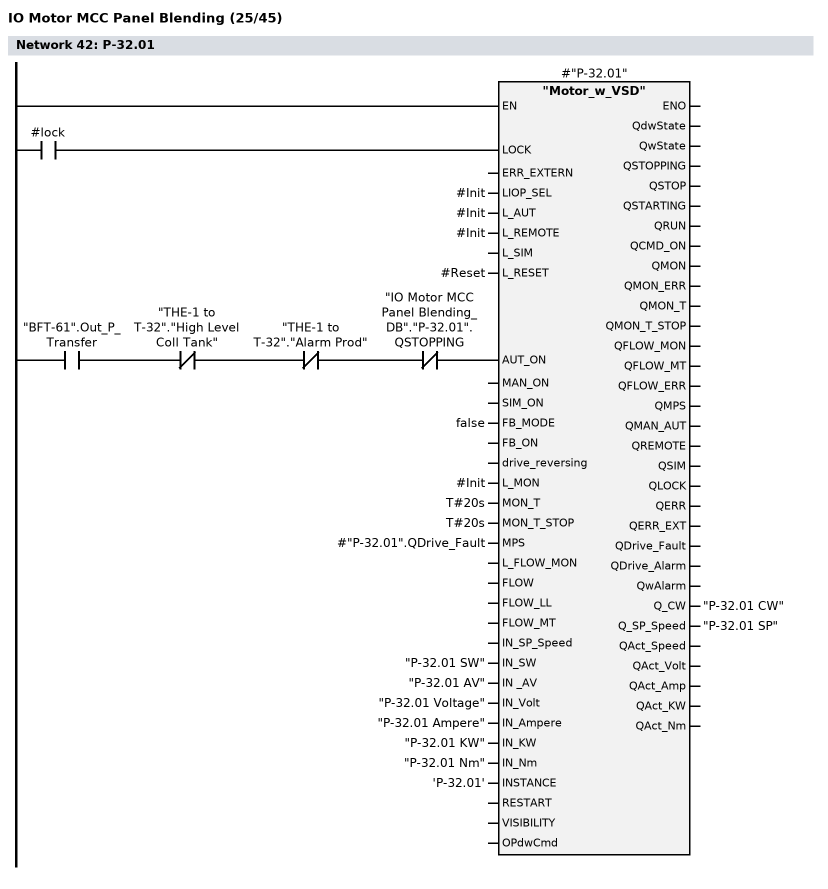
   RUNG wire#powerrail
      #"P-32.01"(LOCK := wire#w1, AUT_ON := wire#w2, ERR_EXTERN :=, LIOP_SEL := #Init, L_AUT := #Init, L_REMOTE := #Init, L_SIM :=, L_RESET := #Reset, MAN_ON :=, SIM_ON :=, FB_MODE := false, FB_ON :=, drive_reversing :=, L_MON := #Init, MON_T := T#20s, MON_T_STOP := T#20s, MPS := #"P-32.01".QDrive_Fault, L_FLOW_MON :=, FLOW :=, FLOW_LL :=, FLOW_MT :=, IN_SP_Speed :=, IN_SW := "P-32.01 SW", "IN _AV" := "P-32.01 AV", IN_Volt := "P-32.01 Voltage", IN_Ampere := "P-32.01 Ampere", IN_KW := "P-32.01 KW", IN_Nm := "P-32.01 Nm", INSTANCE := 'P-32.01', RESTART :=, VISIBILITY :=, OPdwCmd :=, QdwState =>, QwState =>, QSTOPPING =>, QSTOP =>, QSTARTING =>, QRUN =>, QCMD_ON =>, QMON =>, QMON_ERR =>, QMON_T =>, QMON_T_STOP =>, QFLOW_MON =>, QFLOW_MT =>, QFLOW_ERR =>, QMPS =>, QMAN_AUT =>, QREMOTE =>, QSIM =>, QLOCK =>, QERR =>, QERR_EXT =>, QDrive_Fault =>, QDrive_Alarm =>, QwAlarm =>, Q_CW => "P-32.01 CW", Q_SP_Speed => "P-32.01 SP", QAct_Speed =>, QAct_Volt =>, QAct_Amp =>, QAct_KW =>, QAct_Nm =>)
   END_RUNG
   RUNG wire#powerrail
      Contact( #lock )
   END_RUNG wire#w1
   RUNG wire#powerrail
      Contact( "BFT-61".Out_P_Transfer )
      I_Contact( "THE-1 to T-32"."High Level Coll Tank" )
      I_Contact( "THE-1 to T-32"."Alarm Prod" )
      I_Contact( "IO Motor MCC Panel Blending_DB"."P-32.01".QSTOPPING )
   END_RUNG wire#w2
   // the same network as SCL:
   #"P-32.01"(LOCK := #lock,   // "Motor_w_VSD"
              LIOP_SEL := #Init,
              L_AUT := #Init,
              L_REMOTE := #Init,
              L_RESET := #Reset,
              AUT_ON := "BFT-61".Out_P_Transfer AND NOT "THE-1 to T-32"."High Level Coll Tank" AND NOT "THE-1 to T-32"."Alarm Prod" AND NOT "IO Motor MCC Panel Blending_DB"."P-32.01".QSTOPPING,
              FB_MODE := false,
              L_MON := #Init,
              MON_T := T#20s,
              MON_T_STOP := T#20s,
              MPS := #"P-32.01".QDrive_Fault,
              IN_SW := "P-32.01 SW",
              "IN _AV" := "P-32.01 AV",
              IN_Volt := "P-32.01 Voltage",
              IN_Ampere := "P-32.01 Ampere",
              IN_KW := "P-32.01 KW",
              IN_Nm := "P-32.01 Nm",
              INSTANCE := 'P-32.01',
              Q_CW => "P-32.01 CW",
              Q_SP_Speed => "P-32.01 SP");
END_REGION

REGION Network 43: P-32.02
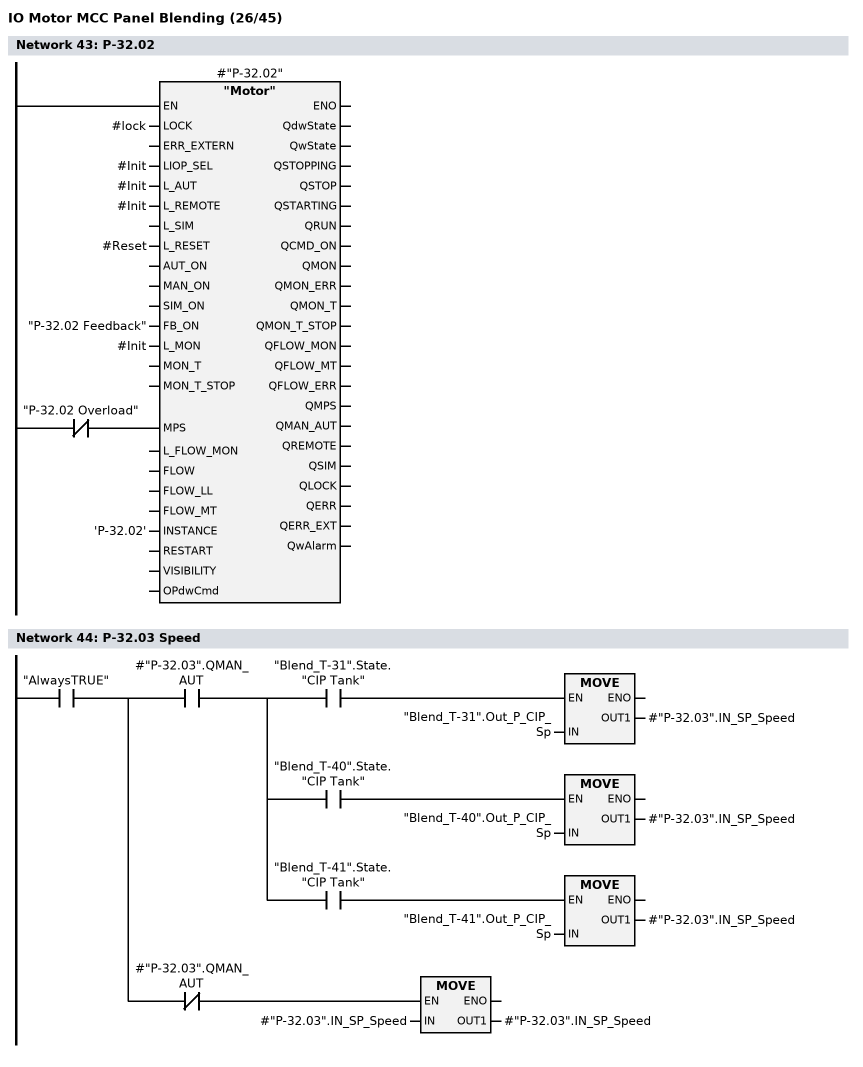
   RUNG wire#powerrail
      #"P-32.02"(MPS := wire#w1, LOCK := #lock, ERR_EXTERN :=, LIOP_SEL := #Init, L_AUT := #Init, L_REMOTE := #Init, L_SIM :=, L_RESET := #Reset, AUT_ON :=, MAN_ON :=, SIM_ON :=, FB_ON := "P-32.02 Feedback", L_MON := #Init, MON_T :=, MON_T_STOP :=, L_FLOW_MON :=, FLOW :=, FLOW_LL :=, FLOW_MT :=, INSTANCE := 'P-32.02', RESTART :=, VISIBILITY :=, OPdwCmd :=, QdwState =>, QwState =>, QSTOPPING =>, QSTOP =>, QSTARTING =>, QRUN =>, QCMD_ON =>, QMON =>, QMON_ERR =>, QMON_T =>, QMON_T_STOP =>, QFLOW_MON =>, QFLOW_MT =>, QFLOW_ERR =>, QMPS =>, QMAN_AUT =>, QREMOTE =>, QSIM =>, QLOCK =>, QERR =>, QERR_EXT =>, QwAlarm =>)
   END_RUNG
   RUNG wire#powerrail
      I_Contact( "P-32.02 Overload" )
   END_RUNG wire#w1
   // the same network as SCL:
   #"P-32.02"(LOCK := #lock,   // "Motor"
              LIOP_SEL := #Init,
              L_AUT := #Init,
              L_REMOTE := #Init,
              L_RESET := #Reset,
              FB_ON := "P-32.02 Feedback",
              L_MON := #Init,
              MPS := NOT "P-32.02 Overload",
              INSTANCE := 'P-32.02');
END_REGION

REGION Network 44: P-32.03 Speed
   RUNG wire#powerrail
      Contact( "AlwaysTRUE" )
      wire#w1
      Contact( #"P-32.03".QMAN_AUT )
      wire#w2
      Contact( "Blend_T-31".State."CIP Tank" )
      Move(in := "Blend_T-31".Out_P_CIP_Sp, out1 => #"P-32.03".IN_SP_Speed)
   END_RUNG
   RUNG wire#w2
      Contact( "Blend_T-40".State."CIP Tank" )
      Move(in := "Blend_T-40".Out_P_CIP_Sp, out1 => #"P-32.03".IN_SP_Speed)
   END_RUNG
   RUNG wire#w2
      Contact( "Blend_T-41".State."CIP Tank" )
      Move(in := "Blend_T-41".Out_P_CIP_Sp, out1 => #"P-32.03".IN_SP_Speed)
   END_RUNG
   RUNG wire#w1
      I_Contact( #"P-32.03".QMAN_AUT )
      Move(in := #"P-32.03".IN_SP_Speed, out1 => #"P-32.03".IN_SP_Speed)
   END_RUNG
   // the same network as SCL:
   #_w1 := "AlwaysTRUE" AND #"P-32.03".QMAN_AUT;
   IF #_w1 AND "Blend_T-31".State."CIP Tank" THEN
       #"P-32.03".IN_SP_Speed := "Blend_T-31".Out_P_CIP_Sp;
   END_IF;
   IF #_w1 AND "Blend_T-40".State."CIP Tank" THEN
       #"P-32.03".IN_SP_Speed := "Blend_T-40".Out_P_CIP_Sp;
   END_IF;
   IF #_w1 AND "Blend_T-41".State."CIP Tank" THEN
       #"P-32.03".IN_SP_Speed := "Blend_T-41".Out_P_CIP_Sp;
   END_IF;
   IF "AlwaysTRUE" AND NOT #"P-32.03".QMAN_AUT THEN #"P-32.03".IN_SP_Speed := #"P-32.03".IN_SP_Speed; END_IF;
END_REGION

REGION Network 45: P-32.03
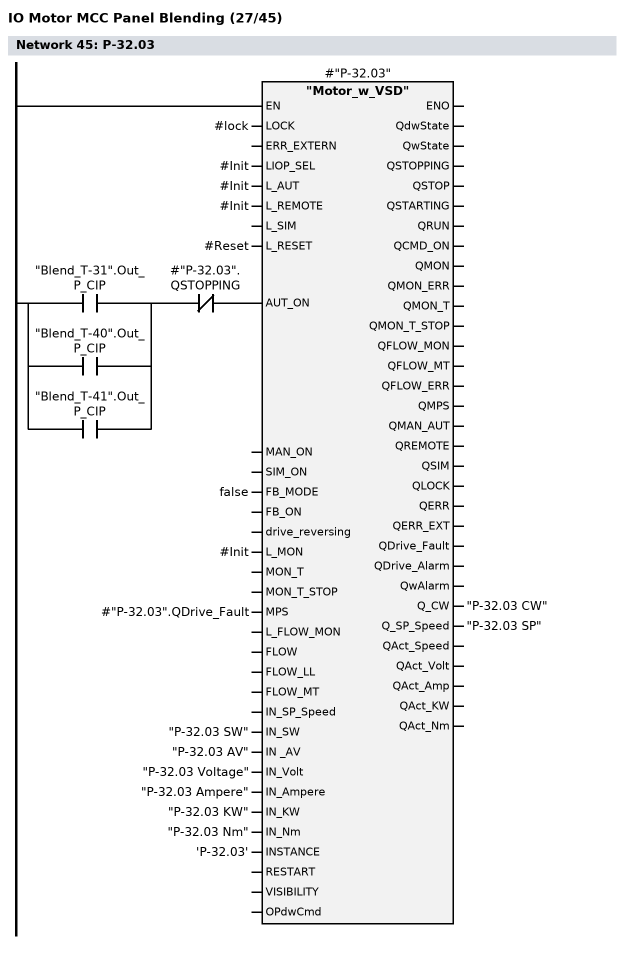
   RUNG wire#powerrail
      #"P-32.03"(AUT_ON := wire#w2, LOCK := #lock, ERR_EXTERN :=, LIOP_SEL := #Init, L_AUT := #Init, L_REMOTE := #Init, L_SIM :=, L_RESET := #Reset, MAN_ON :=, SIM_ON :=, FB_MODE := false, FB_ON :=, drive_reversing :=, L_MON := #Init, MON_T :=, MON_T_STOP :=, MPS := #"P-32.03".QDrive_Fault, L_FLOW_MON :=, FLOW :=, FLOW_LL :=, FLOW_MT :=, IN_SP_Speed :=, IN_SW := "P-32.03 SW", "IN _AV" := "P-32.03 AV", IN_Volt := "P-32.03 Voltage", IN_Ampere := "P-32.03 Ampere", IN_KW := "P-32.03 KW", IN_Nm := "P-32.03 Nm", INSTANCE := 'P-32.03', RESTART :=, VISIBILITY :=, OPdwCmd :=, QdwState =>, QwState =>, QSTOPPING =>, QSTOP =>, QSTARTING =>, QRUN =>, QCMD_ON =>, QMON =>, QMON_ERR =>, QMON_T =>, QMON_T_STOP =>, QFLOW_MON =>, QFLOW_MT =>, QFLOW_ERR =>, QMPS =>, QMAN_AUT =>, QREMOTE =>, QSIM =>, QLOCK =>, QERR =>, QERR_EXT =>, QDrive_Fault =>, QDrive_Alarm =>, QwAlarm =>, Q_CW => "P-32.03 CW", Q_SP_Speed => "P-32.03 SP", QAct_Speed =>, QAct_Volt =>, QAct_Amp =>, QAct_KW =>, QAct_Nm =>)
   END_RUNG
   RUNG wire#powerrail
      Contact( "Blend_T-31".Out_P_CIP )
      wire#w1
      I_Contact( #"P-32.03".QSTOPPING )
   END_RUNG wire#w2
   RUNG wire#powerrail
      Contact( "Blend_T-40".Out_P_CIP )
   END_RUNG wire#w1
   RUNG wire#powerrail
      Contact( "Blend_T-41".Out_P_CIP )
   END_RUNG wire#w1
   // the same network as SCL:
   #"P-32.03"(LOCK := #lock,   // "Motor_w_VSD"
              LIOP_SEL := #Init,
              L_AUT := #Init,
              L_REMOTE := #Init,
              L_RESET := #Reset,
              AUT_ON := ("Blend_T-31".Out_P_CIP OR "Blend_T-40".Out_P_CIP OR "Blend_T-41".Out_P_CIP) AND NOT #"P-32.03".QSTOPPING,
              FB_MODE := false,
              L_MON := #Init,
              MPS := #"P-32.03".QDrive_Fault,
              IN_SW := "P-32.03 SW",
              "IN _AV" := "P-32.03 AV",
              IN_Volt := "P-32.03 Voltage",
              IN_Ampere := "P-32.03 Ampere",
              IN_KW := "P-32.03 KW",
              IN_Nm := "P-32.03 Nm",
              INSTANCE := 'P-32.03',
              Q_CW => "P-32.03 CW",
              Q_SP_Speed => "P-32.03 SP");
END_REGION

REGION Network 46: P-32 Circulation (P-32.04)
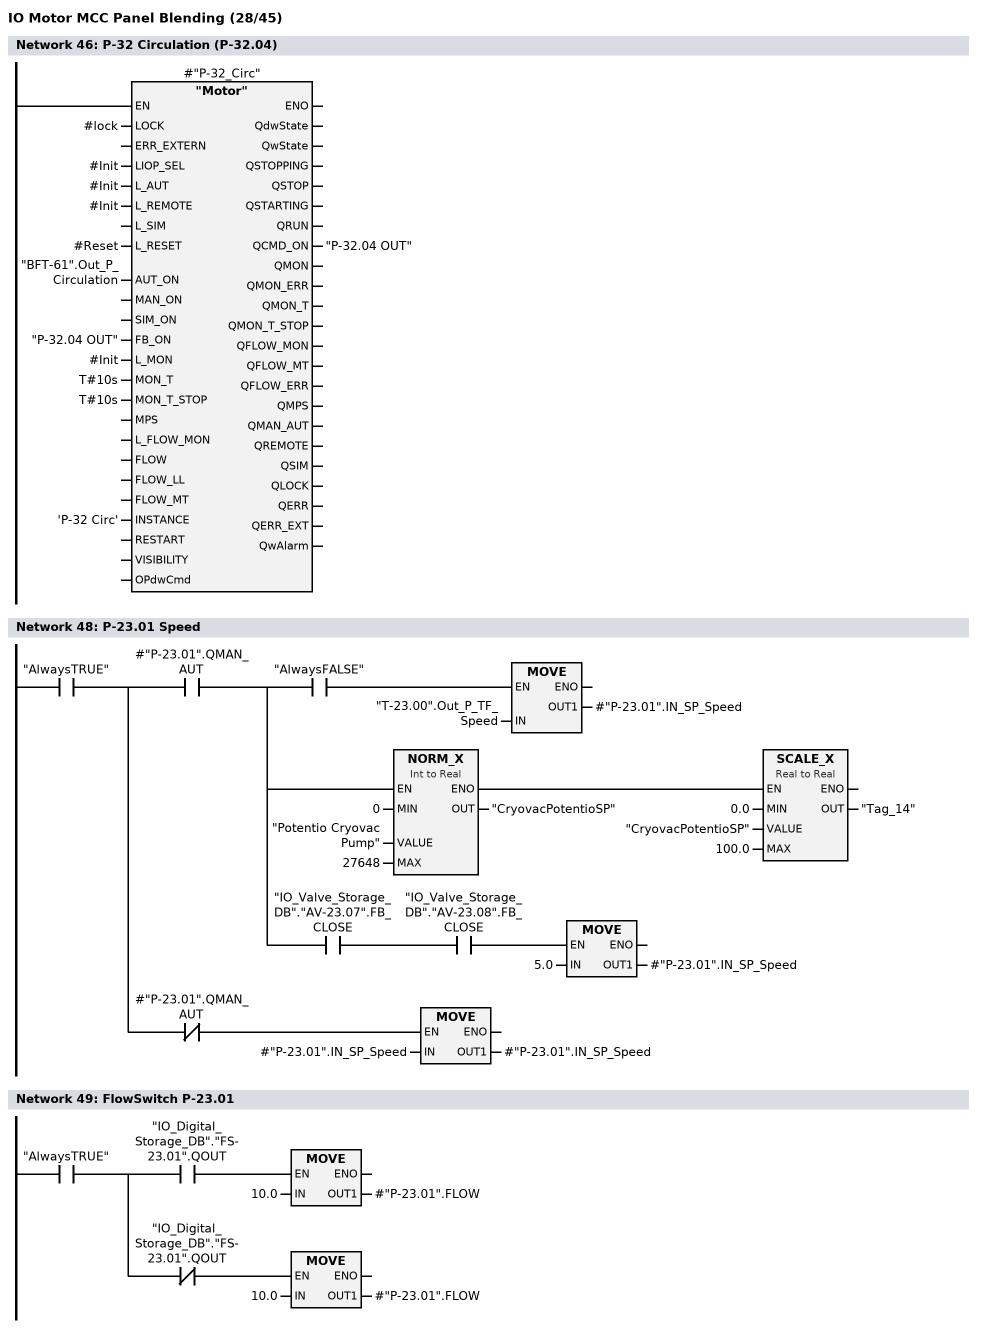
   RUNG wire#powerrail
      #"P-32_Circ"(LOCK := #lock, ERR_EXTERN :=, LIOP_SEL := #Init, L_AUT := #Init, L_REMOTE := #Init, L_SIM :=, L_RESET := #Reset, AUT_ON := "BFT-61".Out_P_Circulation, MAN_ON :=, SIM_ON :=, FB_ON := "P-32.04 OUT", L_MON := #Init, MON_T := T#10s, MON_T_STOP := T#10s, MPS :=, L_FLOW_MON :=, FLOW :=, FLOW_LL :=, FLOW_MT :=, INSTANCE := 'P-32 Circ', RESTART :=, VISIBILITY :=, OPdwCmd :=, QdwState =>, QwState =>, QSTOPPING =>, QSTOP =>, QSTARTING =>, QRUN =>, QCMD_ON => "P-32.04 OUT", QMON =>, QMON_ERR =>, QMON_T =>, QMON_T_STOP =>, QFLOW_MON =>, QFLOW_MT =>, QFLOW_ERR =>, QMPS =>, QMAN_AUT =>, QREMOTE =>, QSIM =>, QLOCK =>, QERR =>, QERR_EXT =>, QwAlarm =>)
   END_RUNG
   // the same network as SCL:
   #"P-32_Circ"(LOCK := #lock,   // "Motor"
                LIOP_SEL := #Init,
                L_AUT := #Init,
                L_REMOTE := #Init,
                L_RESET := #Reset,
                AUT_ON := "BFT-61".Out_P_Circulation,
                FB_ON := "P-32.04 OUT",
                L_MON := #Init,
                MON_T := T#10s,
                MON_T_STOP := T#10s,
                INSTANCE := 'P-32 Circ',
                QCMD_ON => "P-32.04 OUT");
END_REGION

REGION Network 48: P-23.01 Speed
   RUNG wire#powerrail
      Contact( "AlwaysTRUE" )
      wire#w1
      Contact( #"P-23.01".QMAN_AUT )
      wire#w2
      Contact( "AlwaysFALSE" )
      Move(in := "T-23.00".Out_P_TF_Speed, out1 => #"P-23.01".IN_SP_Speed)
   END_RUNG
   RUNG wire#w2
      { S7_Templates := "[SrcType := Int, DestType := Real]" } Normalize(min := 0, value := "Potentio Cryovac Pump", max := 27648, out => "CryovacPotentioSP")
      { S7_Templates := "[SrcType := Real, DestType := Real]" } Scale(min := 0.0, value := "CryovacPotentioSP", max := 100.0, out => "Tag_14")
   END_RUNG
   RUNG wire#w2
      Contact( "IO_Valve_Storage_DB"."AV-23.07".FB_CLOSE )
      Contact( "IO_Valve_Storage_DB"."AV-23.08".FB_CLOSE )
      Move(in := 5.0, out1 => #"P-23.01".IN_SP_Speed)
   END_RUNG
   RUNG wire#w1
      I_Contact( #"P-23.01".QMAN_AUT )
      Move(in := #"P-23.01".IN_SP_Speed, out1 => #"P-23.01".IN_SP_Speed)
   END_RUNG
   // the same network as SCL:
   #_w1 := "AlwaysTRUE" AND #"P-23.01".QMAN_AUT;
   IF #_w1 AND "AlwaysFALSE" THEN #"P-23.01".IN_SP_Speed := "T-23.00".Out_P_TF_Speed; END_IF;
   IF #_w1 THEN
       "CryovacPotentioSP" := NORM_X(MIN := 0, VALUE := "Potentio Cryovac Pump", MAX := 27648);
       "Tag_14" := SCALE_X(MIN := 0.0, VALUE := "CryovacPotentioSP", MAX := 100.0);
   END_IF;
   IF #_w1 AND "IO_Valve_Storage_DB"."AV-23.07".FB_CLOSE AND "IO_Valve_Storage_DB"."AV-23.08".FB_CLOSE THEN
       #"P-23.01".IN_SP_Speed := 5.0;
   END_IF;
   IF "AlwaysTRUE" AND NOT #"P-23.01".QMAN_AUT THEN #"P-23.01".IN_SP_Speed := #"P-23.01".IN_SP_Speed; END_IF;
END_REGION

REGION Network 49: FlowSwitch P-23.01
   RUNG wire#powerrail
      Contact( "AlwaysTRUE" )
      wire#w1
      Contact( "IO_Digital_Storage_DB"."FS-23.01".QOUT )
      Move(in := 10.0, out1 => #"P-23.01".FLOW)
   END_RUNG
   RUNG wire#w1
      I_Contact( "IO_Digital_Storage_DB"."FS-23.01".QOUT )
      Move(in := 10.0, out1 => #"P-23.01".FLOW)
   END_RUNG
   // the same network as SCL:
   IF "AlwaysTRUE" AND "IO_Digital_Storage_DB"."FS-23.01".QOUT THEN #"P-23.01".FLOW := 10.0; END_IF;
   IF "AlwaysTRUE" AND NOT "IO_Digital_Storage_DB"."FS-23.01".QOUT THEN #"P-23.01".FLOW := 10.0; END_IF;
END_REGION

REGION Network 50: P-23.01
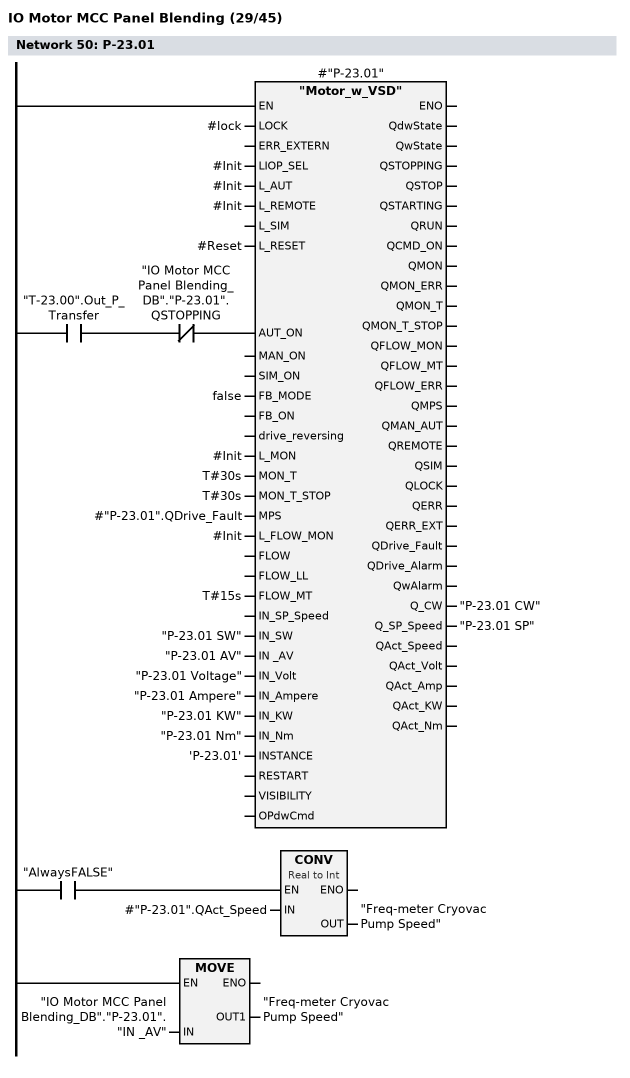
   RUNG wire#powerrail
      #"P-23.01"(AUT_ON := wire#w1, LOCK := #lock, ERR_EXTERN :=, LIOP_SEL := #Init, L_AUT := #Init, L_REMOTE := #Init, L_SIM :=, L_RESET := #Reset, MAN_ON :=, SIM_ON :=, FB_MODE := false, FB_ON :=, drive_reversing :=, L_MON := #Init, MON_T := T#30s, MON_T_STOP := T#30s, MPS := #"P-23.01".QDrive_Fault, L_FLOW_MON := #Init, FLOW :=, FLOW_LL :=, FLOW_MT := T#15s, IN_SP_Speed :=, IN_SW := "P-23.01 SW", "IN _AV" := "P-23.01 AV", IN_Volt := "P-23.01 Voltage", IN_Ampere := "P-23.01 Ampere", IN_KW := "P-23.01 KW", IN_Nm := "P-23.01 Nm", INSTANCE := 'P-23.01', RESTART :=, VISIBILITY :=, OPdwCmd :=, QdwState =>, QwState =>, QSTOPPING =>, QSTOP =>, QSTARTING =>, QRUN =>, QCMD_ON =>, QMON =>, QMON_ERR =>, QMON_T =>, QMON_T_STOP =>, QFLOW_MON =>, QFLOW_MT =>, QFLOW_ERR =>, QMPS =>, QMAN_AUT =>, QREMOTE =>, QSIM =>, QLOCK =>, QERR =>, QERR_EXT =>, QDrive_Fault =>, QDrive_Alarm =>, QwAlarm =>, Q_CW => "P-23.01 CW", Q_SP_Speed => "P-23.01 SP", QAct_Speed =>, QAct_Volt =>, QAct_Amp =>, QAct_KW =>, QAct_Nm =>)
   END_RUNG
   RUNG wire#powerrail
      Contact( "T-23.00".Out_P_Transfer )
      I_Contact( "IO Motor MCC Panel Blending_DB"."P-23.01".QSTOPPING )
   END_RUNG wire#w1
   RUNG wire#powerrail
      Contact( "AlwaysFALSE" )
      { S7_Templates := "[SrcType := Real, DestType := Int]" } Convert(in := #"P-23.01".QAct_Speed, out => "Freq-meter Cryovac Pump Speed")
   END_RUNG
   RUNG wire#powerrail
      Move(in := "IO Motor MCC Panel Blending_DB"."P-23.01"."IN _AV", out1 => "Freq-meter Cryovac Pump Speed")
   END_RUNG
   // the same network as SCL:
   #"P-23.01"(LOCK := #lock,   // "Motor_w_VSD"
              LIOP_SEL := #Init,
              L_AUT := #Init,
              L_REMOTE := #Init,
              L_RESET := #Reset,
              AUT_ON := "T-23.00".Out_P_Transfer AND NOT "IO Motor MCC Panel Blending_DB"."P-23.01".QSTOPPING,
              FB_MODE := false,
              L_MON := #Init,
              MON_T := T#30s,
              MON_T_STOP := T#30s,
              MPS := #"P-23.01".QDrive_Fault,
              L_FLOW_MON := #Init,
              FLOW_MT := T#15s,
              IN_SW := "P-23.01 SW",
              "IN _AV" := "P-23.01 AV",
              IN_Volt := "P-23.01 Voltage",
              IN_Ampere := "P-23.01 Ampere",
              IN_KW := "P-23.01 KW",
              IN_Nm := "P-23.01 Nm",
              INSTANCE := 'P-23.01',
              Q_CW => "P-23.01 CW",
              Q_SP_Speed => "P-23.01 SP");
   IF "AlwaysFALSE" THEN "Freq-meter Cryovac Pump Speed" := REAL_TO_INT(#"P-23.01".QAct_Speed); END_IF;
   "Freq-meter Cryovac Pump Speed" := "IO Motor MCC Panel Blending_DB"."P-23.01"."IN _AV";
END_REGION

REGION Network 52: P-24.01 Speed
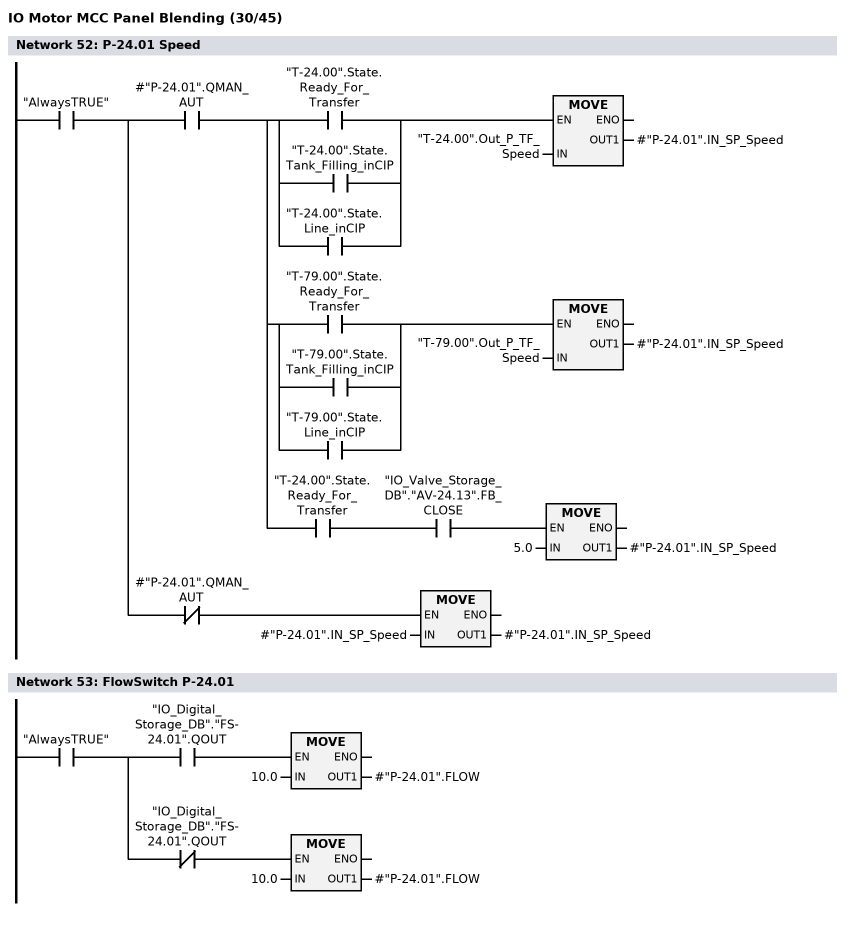
   RUNG wire#powerrail
      Contact( "AlwaysTRUE" )
      wire#w1
      Contact( #"P-24.01".QMAN_AUT )
      wire#w2
      Contact( "T-24.00".State.Ready_For_Transfer )
      wire#w3
      Move(in := "T-24.00".Out_P_TF_Speed, out1 => #"P-24.01".IN_SP_Speed)
   END_RUNG
   RUNG wire#w2
      Contact( "T-24.00".State.Tank_Filling_inCIP )
   END_RUNG wire#w3
   RUNG wire#w2
      Contact( "T-24.00".State.Line_inCIP )
   END_RUNG wire#w3
   RUNG wire#w2
      Contact( "T-79.00".State.Ready_For_Transfer )
      wire#w4
      Move(in := "T-79.00".Out_P_TF_Speed, out1 => #"P-24.01".IN_SP_Speed)
   END_RUNG
   RUNG wire#w2
      Contact( "T-79.00".State.Tank_Filling_inCIP )
   END_RUNG wire#w4
   RUNG wire#w2
      Contact( "T-79.00".State.Line_inCIP )
   END_RUNG wire#w4
   RUNG wire#w2
      Contact( "T-24.00".State.Ready_For_Transfer )
      Contact( "IO_Valve_Storage_DB"."AV-24.13".FB_CLOSE )
      Move(in := 5.0, out1 => #"P-24.01".IN_SP_Speed)
   END_RUNG
   RUNG wire#w1
      I_Contact( #"P-24.01".QMAN_AUT )
      Move(in := #"P-24.01".IN_SP_Speed, out1 => #"P-24.01".IN_SP_Speed)
   END_RUNG
   // the same network as SCL:
   #_w1 := "AlwaysTRUE" AND #"P-24.01".QMAN_AUT;
   IF #_w1 AND ("T-24.00".State.Ready_For_Transfer OR "T-24.00".State.Tank_Filling_inCIP OR "T-24.00".State.Line_inCIP) THEN
       #"P-24.01".IN_SP_Speed := "T-24.00".Out_P_TF_Speed;
   END_IF;
   IF #_w1 AND ("T-79.00".State.Ready_For_Transfer OR "T-79.00".State.Tank_Filling_inCIP OR "T-79.00".State.Line_inCIP) THEN
       #"P-24.01".IN_SP_Speed := "T-79.00".Out_P_TF_Speed;
   END_IF;
   IF #_w1 AND "T-24.00".State.Ready_For_Transfer AND "IO_Valve_Storage_DB"."AV-24.13".FB_CLOSE THEN
       #"P-24.01".IN_SP_Speed := 5.0;
   END_IF;
   IF "AlwaysTRUE" AND NOT #"P-24.01".QMAN_AUT THEN #"P-24.01".IN_SP_Speed := #"P-24.01".IN_SP_Speed; END_IF;
END_REGION

REGION Network 53: FlowSwitch P-24.01
   RUNG wire#powerrail
      Contact( "AlwaysTRUE" )
      wire#w1
      Contact( "IO_Digital_Storage_DB"."FS-24.01".QOUT )
      Move(in := 10.0, out1 => #"P-24.01".FLOW)
   END_RUNG
   RUNG wire#w1
      I_Contact( "IO_Digital_Storage_DB"."FS-24.01".QOUT )
      Move(in := 10.0, out1 => #"P-24.01".FLOW)
   END_RUNG
   // the same network as SCL:
   IF "AlwaysTRUE" AND "IO_Digital_Storage_DB"."FS-24.01".QOUT THEN #"P-24.01".FLOW := 10.0; END_IF;
   IF "AlwaysTRUE" AND NOT "IO_Digital_Storage_DB"."FS-24.01".QOUT THEN #"P-24.01".FLOW := 10.0; END_IF;
END_REGION

REGION Network 54: P-24.01
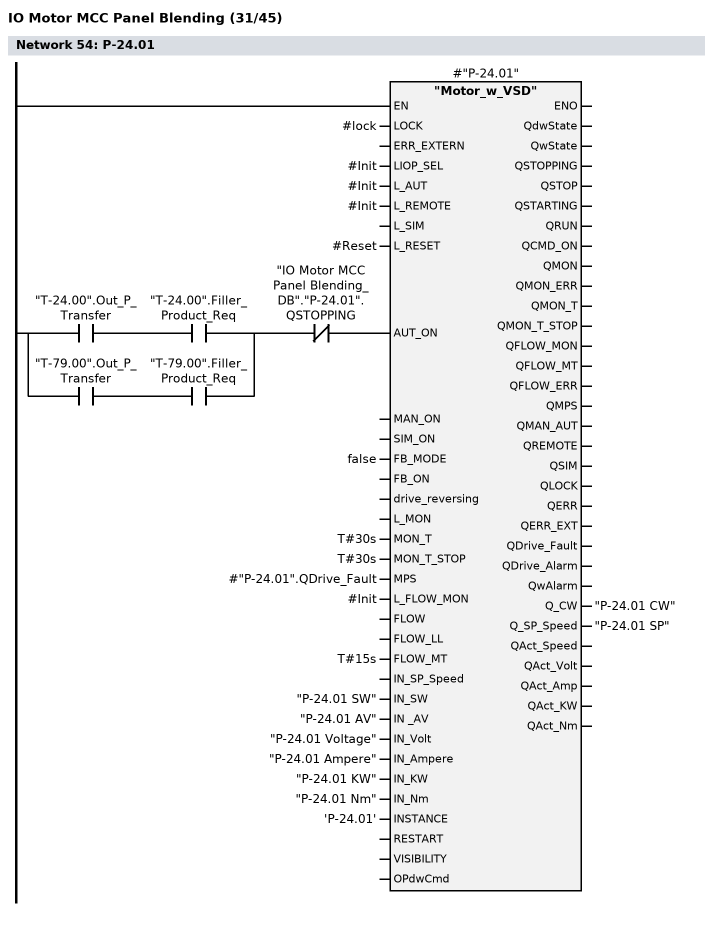
   RUNG wire#powerrail
      #"P-24.01"(AUT_ON := wire#w2, LOCK := #lock, ERR_EXTERN :=, LIOP_SEL := #Init, L_AUT := #Init, L_REMOTE := #Init, L_SIM :=, L_RESET := #Reset, MAN_ON :=, SIM_ON :=, FB_MODE := false, FB_ON :=, drive_reversing :=, L_MON :=, MON_T := T#30s, MON_T_STOP := T#30s, MPS := #"P-24.01".QDrive_Fault, L_FLOW_MON := #Init, FLOW :=, FLOW_LL :=, FLOW_MT := T#15s, IN_SP_Speed :=, IN_SW := "P-24.01 SW", "IN _AV" := "P-24.01 AV", IN_Volt := "P-24.01 Voltage", IN_Ampere := "P-24.01 Ampere", IN_KW := "P-24.01 KW", IN_Nm := "P-24.01 Nm", INSTANCE := 'P-24.01', RESTART :=, VISIBILITY :=, OPdwCmd :=, QdwState =>, QwState =>, QSTOPPING =>, QSTOP =>, QSTARTING =>, QRUN =>, QCMD_ON =>, QMON =>, QMON_ERR =>, QMON_T =>, QMON_T_STOP =>, QFLOW_MON =>, QFLOW_MT =>, QFLOW_ERR =>, QMPS =>, QMAN_AUT =>, QREMOTE =>, QSIM =>, QLOCK =>, QERR =>, QERR_EXT =>, QDrive_Fault =>, QDrive_Alarm =>, QwAlarm =>, Q_CW => "P-24.01 CW", Q_SP_Speed => "P-24.01 SP", QAct_Speed =>, QAct_Volt =>, QAct_Amp =>, QAct_KW =>, QAct_Nm =>)
   END_RUNG
   RUNG wire#powerrail
      Contact( "T-24.00".Out_P_Transfer )
      Contact( "T-24.00".Filler_Product_Req )
      wire#w1
      I_Contact( "IO Motor MCC Panel Blending_DB"."P-24.01".QSTOPPING )
   END_RUNG wire#w2
   RUNG wire#powerrail
      Contact( "T-79.00".Out_P_Transfer )
      Contact( "T-79.00".Filler_Product_Req )
   END_RUNG wire#w1
   // the same network as SCL:
   #"P-24.01"(LOCK := #lock,   // "Motor_w_VSD"
              LIOP_SEL := #Init,
              L_AUT := #Init,
              L_REMOTE := #Init,
              L_RESET := #Reset,
              AUT_ON := (("T-24.00".Out_P_Transfer AND "T-24.00".Filler_Product_Req) OR ("T-79.00".Out_P_Transfer AND "T-79.00".Filler_Product_Req)) AND NOT "IO Motor MCC Panel Blending_DB"."P-24.01".QSTOPPING,
              FB_MODE := false,
              MON_T := T#30s,
              MON_T_STOP := T#30s,
              MPS := #"P-24.01".QDrive_Fault,
              L_FLOW_MON := #Init,
              FLOW_MT := T#15s,
              IN_SW := "P-24.01 SW",
              "IN _AV" := "P-24.01 AV",
              IN_Volt := "P-24.01 Voltage",
              IN_Ampere := "P-24.01 Ampere",
              IN_KW := "P-24.01 KW",
              IN_Nm := "P-24.01 Nm",
              INSTANCE := 'P-24.01',
              Q_CW => "P-24.01 CW",
              Q_SP_Speed => "P-24.01 SP");
END_REGION

REGION Network 55: P-24.02
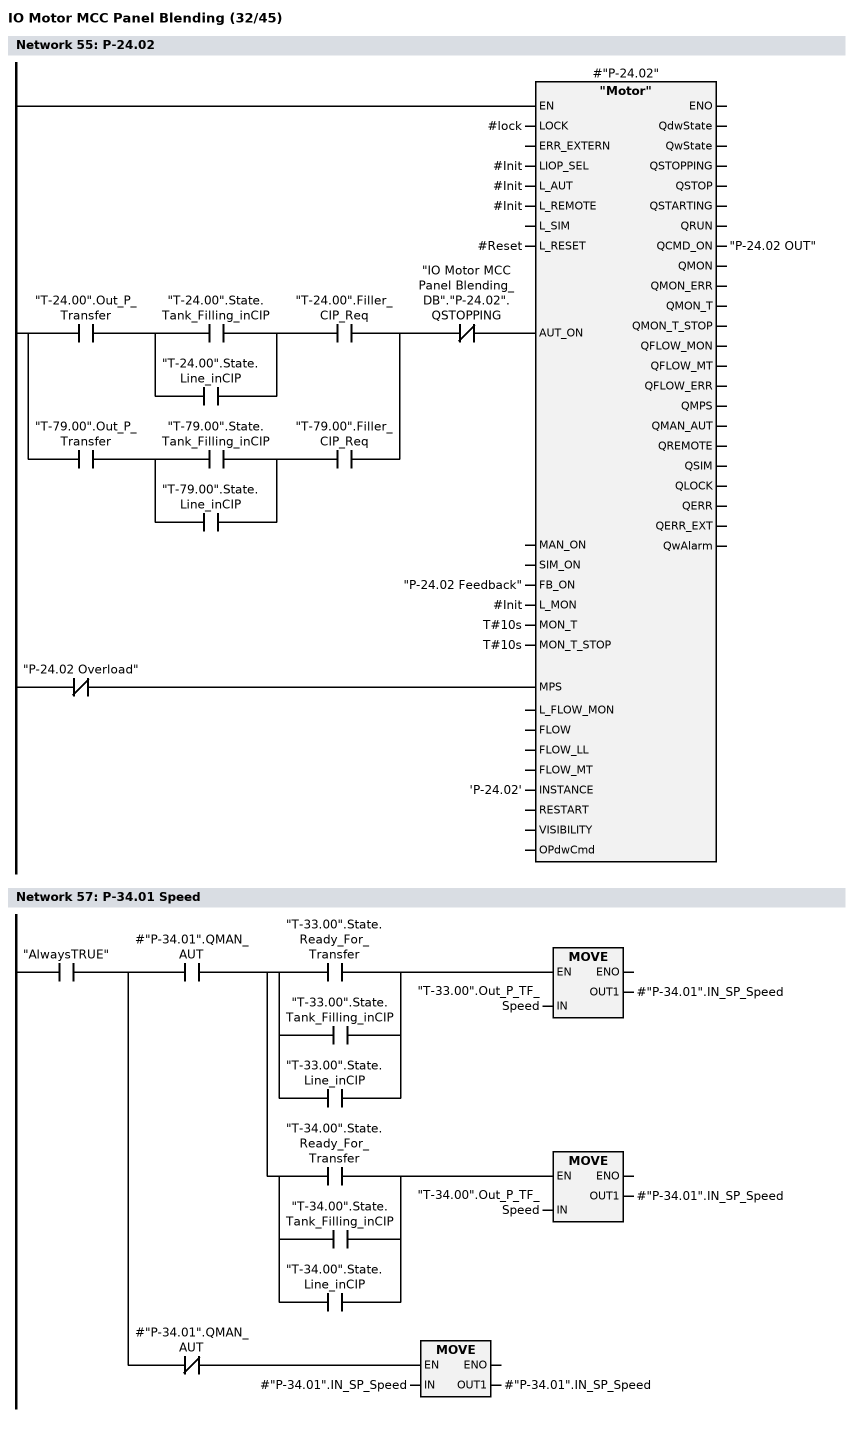
   RUNG wire#powerrail
      #"P-24.02"(AUT_ON := wire#w6, MPS := wire#w7, LOCK := #lock, ERR_EXTERN :=, LIOP_SEL := #Init, L_AUT := #Init, L_REMOTE := #Init, L_SIM :=, L_RESET := #Reset, MAN_ON :=, SIM_ON :=, FB_ON := "P-24.02 Feedback", L_MON := #Init, MON_T := T#10s, MON_T_STOP := T#10s, L_FLOW_MON :=, FLOW :=, FLOW_LL :=, FLOW_MT :=, INSTANCE := 'P-24.02', RESTART :=, VISIBILITY :=, OPdwCmd :=, QdwState =>, QwState =>, QSTOPPING =>, QSTOP =>, QSTARTING =>, QRUN =>, QCMD_ON => "P-24.02 OUT", QMON =>, QMON_ERR =>, QMON_T =>, QMON_T_STOP =>, QFLOW_MON =>, QFLOW_MT =>, QFLOW_ERR =>, QMPS =>, QMAN_AUT =>, QREMOTE =>, QSIM =>, QLOCK =>, QERR =>, QERR_EXT =>, QwAlarm =>)
   END_RUNG
   RUNG wire#powerrail
      Contact( "T-24.00".Out_P_Transfer )
      wire#w1
      Contact( "T-24.00".State.Tank_Filling_inCIP )
      wire#w2
      Contact( "T-24.00".Filler_CIP_Req )
      wire#w3
      I_Contact( "IO Motor MCC Panel Blending_DB"."P-24.02".QSTOPPING )
   END_RUNG wire#w6
   RUNG wire#w1
      Contact( "T-24.00".State.Line_inCIP )
   END_RUNG wire#w2
   RUNG wire#powerrail
      Contact( "T-79.00".Out_P_Transfer )
      wire#w4
      Contact( "T-79.00".State.Tank_Filling_inCIP )
      wire#w5
      Contact( "T-79.00".Filler_CIP_Req )
   END_RUNG wire#w3
   RUNG wire#w4
      Contact( "T-79.00".State.Line_inCIP )
   END_RUNG wire#w5
   RUNG wire#powerrail
      I_Contact( "P-24.02 Overload" )
   END_RUNG wire#w7
   // the same network as SCL:
   #"P-24.02"(LOCK := #lock,   // "Motor"
              LIOP_SEL := #Init,
              L_AUT := #Init,
              L_REMOTE := #Init,
              L_RESET := #Reset,
              AUT_ON := (("T-24.00".Out_P_Transfer AND ("T-24.00".State.Tank_Filling_inCIP OR "T-24.00".State.Line_inCIP) AND "T-24.00".Filler_CIP_Req) OR ("T-79.00".Out_P_Transfer AND ("T-79.00".State.Tank_Filling_inCIP OR "T-79.00".State.Line_inCIP) AND "T-79.00".Filler_CIP_Req)) AND NOT "IO Motor MCC Panel Blending_DB"."P-24.02".QSTOPPING,
              FB_ON := "P-24.02 Feedback",
              L_MON := #Init,
              MON_T := T#10s,
              MON_T_STOP := T#10s,
              MPS := NOT "P-24.02 Overload",
              INSTANCE := 'P-24.02',
              QCMD_ON => "P-24.02 OUT");
END_REGION

REGION Network 57: P-34.01 Speed
   RUNG wire#powerrail
      Contact( "AlwaysTRUE" )
      wire#w1
      Contact( #"P-34.01".QMAN_AUT )
      wire#w2
      Contact( "T-33.00".State.Ready_For_Transfer )
      wire#w3
      Move(in := "T-33.00".Out_P_TF_Speed, out1 => #"P-34.01".IN_SP_Speed)
   END_RUNG
   RUNG wire#w2
      Contact( "T-33.00".State.Tank_Filling_inCIP )
   END_RUNG wire#w3
   RUNG wire#w2
      Contact( "T-33.00".State.Line_inCIP )
   END_RUNG wire#w3
   RUNG wire#w2
      Contact( "T-34.00".State.Ready_For_Transfer )
      wire#w4
      Move(in := "T-34.00".Out_P_TF_Speed, out1 => #"P-34.01".IN_SP_Speed)
   END_RUNG
   RUNG wire#w2
      Contact( "T-34.00".State.Tank_Filling_inCIP )
   END_RUNG wire#w4
   RUNG wire#w2
      Contact( "T-34.00".State.Line_inCIP )
   END_RUNG wire#w4
   RUNG wire#w1
      I_Contact( #"P-34.01".QMAN_AUT )
      Move(in := #"P-34.01".IN_SP_Speed, out1 => #"P-34.01".IN_SP_Speed)
   END_RUNG
   // the same network as SCL:
   #_w1 := "AlwaysTRUE" AND #"P-34.01".QMAN_AUT;
   IF #_w1 AND ("T-33.00".State.Ready_For_Transfer OR "T-33.00".State.Tank_Filling_inCIP OR "T-33.00".State.Line_inCIP) THEN
       #"P-34.01".IN_SP_Speed := "T-33.00".Out_P_TF_Speed;
   END_IF;
   IF #_w1 AND ("T-34.00".State.Ready_For_Transfer OR "T-34.00".State.Tank_Filling_inCIP OR "T-34.00".State.Line_inCIP) THEN
       #"P-34.01".IN_SP_Speed := "T-34.00".Out_P_TF_Speed;
   END_IF;
   IF "AlwaysTRUE" AND NOT #"P-34.01".QMAN_AUT THEN #"P-34.01".IN_SP_Speed := #"P-34.01".IN_SP_Speed; END_IF;
END_REGION

REGION Network 58: FlowSwitch P-34.01
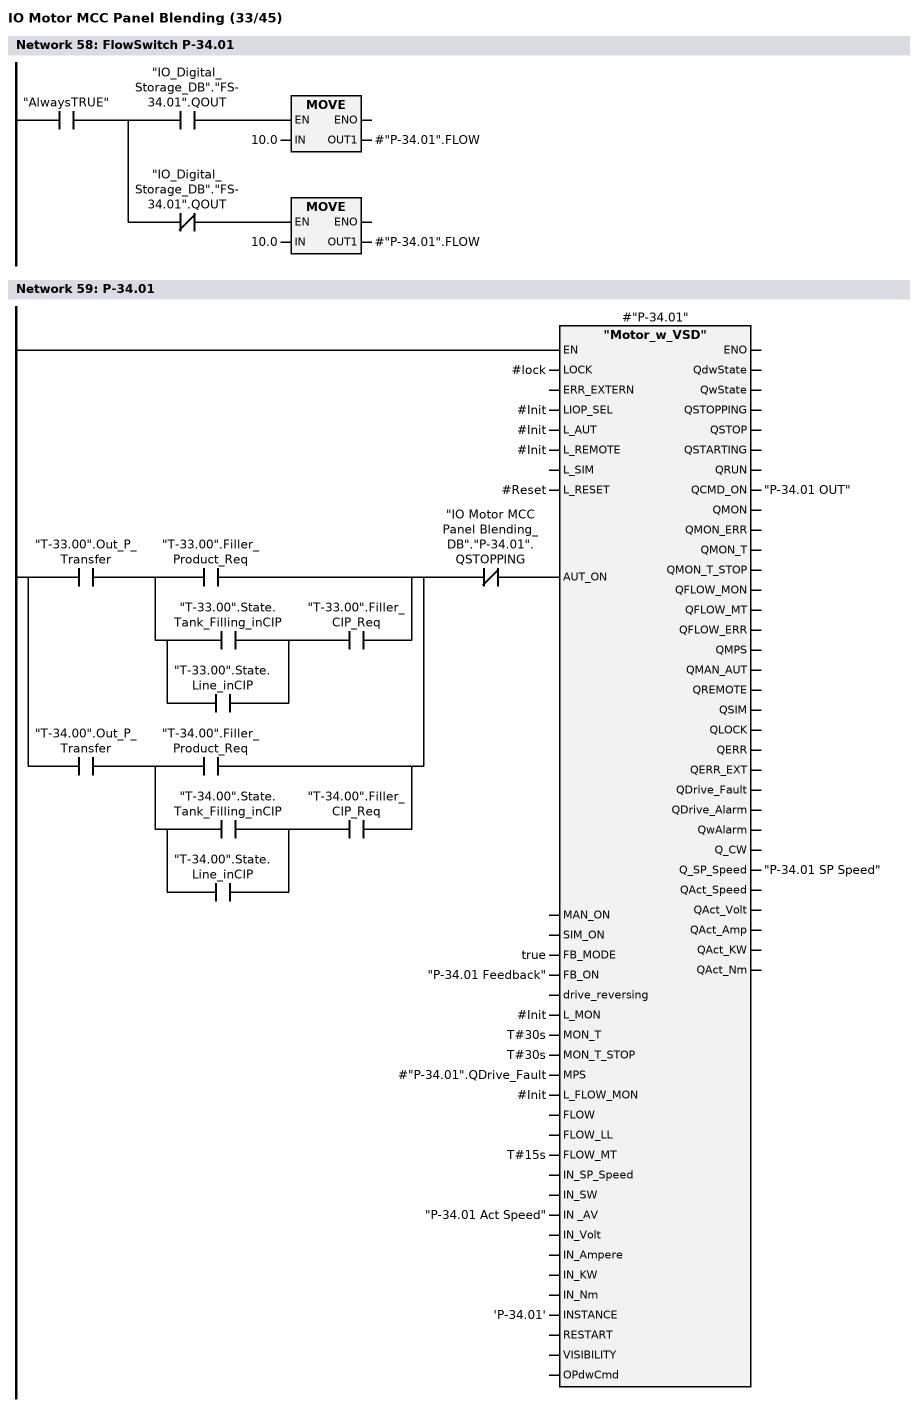
   RUNG wire#powerrail
      Contact( "AlwaysTRUE" )
      wire#w1
      Contact( "IO_Digital_Storage_DB"."FS-34.01".QOUT )
      Move(in := 10.0, out1 => #"P-34.01".FLOW)
   END_RUNG
   RUNG wire#w1
      I_Contact( "IO_Digital_Storage_DB"."FS-34.01".QOUT )
      Move(in := 10.0, out1 => #"P-34.01".FLOW)
   END_RUNG
   // the same network as SCL:
   IF "AlwaysTRUE" AND "IO_Digital_Storage_DB"."FS-34.01".QOUT THEN #"P-34.01".FLOW := 10.0; END_IF;
   IF "AlwaysTRUE" AND NOT "IO_Digital_Storage_DB"."FS-34.01".QOUT THEN #"P-34.01".FLOW := 10.0; END_IF;
END_REGION

REGION Network 59: P-34.01
   RUNG wire#powerrail
      #"P-34.01"(AUT_ON := wire#w6, LOCK := #lock, ERR_EXTERN :=, LIOP_SEL := #Init, L_AUT := #Init, L_REMOTE := #Init, L_SIM :=, L_RESET := #Reset, MAN_ON :=, SIM_ON :=, FB_MODE := true, FB_ON := "P-34.01 Feedback", drive_reversing :=, L_MON := #Init, MON_T := T#30s, MON_T_STOP := T#30s, MPS := #"P-34.01".QDrive_Fault, L_FLOW_MON := #Init, FLOW :=, FLOW_LL :=, FLOW_MT := T#15s, IN_SP_Speed :=, IN_SW :=, "IN _AV" := "P-34.01 Act Speed", IN_Volt :=, IN_Ampere :=, IN_KW :=, IN_Nm :=, INSTANCE := 'P-34.01', RESTART :=, VISIBILITY :=, OPdwCmd :=, QdwState =>, QwState =>, QSTOPPING =>, QSTOP =>, QSTARTING =>, QRUN =>, QCMD_ON => "P-34.01 OUT", QMON =>, QMON_ERR =>, QMON_T =>, QMON_T_STOP =>, QFLOW_MON =>, QFLOW_MT =>, QFLOW_ERR =>, QMPS =>, QMAN_AUT =>, QREMOTE =>, QSIM =>, QLOCK =>, QERR =>, QERR_EXT =>, QDrive_Fault =>, QDrive_Alarm =>, QwAlarm =>, Q_CW =>, Q_SP_Speed => "P-34.01 SP Speed", QAct_Speed =>, QAct_Volt =>, QAct_Amp =>, QAct_KW =>, QAct_Nm =>)
   END_RUNG
   RUNG wire#powerrail
      Contact( "T-33.00".Out_P_Transfer )
      wire#w1
      Contact( "T-33.00".Filler_Product_Req )
      wire#w2
      I_Contact( "IO Motor MCC Panel Blending_DB"."P-34.01".QSTOPPING )
   END_RUNG wire#w6
   RUNG wire#w1
      Contact( "T-33.00".State.Tank_Filling_inCIP )
      wire#w3
      Contact( "T-33.00".Filler_CIP_Req )
   END_RUNG wire#w2
   RUNG wire#w1
      Contact( "T-33.00".State.Line_inCIP )
   END_RUNG wire#w3
   RUNG wire#powerrail
      Contact( "T-34.00".Out_P_Transfer )
      wire#w4
      Contact( "T-34.00".Filler_Product_Req )
   END_RUNG wire#w2
   RUNG wire#w4
      Contact( "T-34.00".State.Tank_Filling_inCIP )
      wire#w5
      Contact( "T-34.00".Filler_CIP_Req )
   END_RUNG wire#w2
   RUNG wire#w4
      Contact( "T-34.00".State.Line_inCIP )
   END_RUNG wire#w5
   // the same network as SCL:
   #"P-34.01"(LOCK := #lock,   // "Motor_w_VSD"
              LIOP_SEL := #Init,
              L_AUT := #Init,
              L_REMOTE := #Init,
              L_RESET := #Reset,
              AUT_ON := (("T-33.00".Out_P_Transfer AND ("T-33.00".Filler_Product_Req OR (("T-33.00".State.Tank_Filling_inCIP OR "T-33.00".State.Line_inCIP) AND "T-33.00".Filler_CIP_Req))) OR ("T-34.00".Out_P_Transfer AND ("T-34.00".Filler_Product_Req OR (("T-34.00".State.Tank_Filling_inCIP OR "T-34.00".State.Line_inCIP) AND "T-34.00".Filler_CIP_Req)))) AND NOT "IO Motor MCC Panel Blending_DB"."P-34.01".QSTOPPING,
              FB_MODE := true,
              FB_ON := "P-34.01 Feedback",
              L_MON := #Init,
              MON_T := T#30s,
              MON_T_STOP := T#30s,
              MPS := #"P-34.01".QDrive_Fault,
              L_FLOW_MON := #Init,
              FLOW_MT := T#15s,
              "IN _AV" := "P-34.01 Act Speed",
              INSTANCE := 'P-34.01',
              QCMD_ON => "P-34.01 OUT",
              Q_SP_Speed => "P-34.01 SP Speed");
END_REGION

REGION Network 60: P-34.02
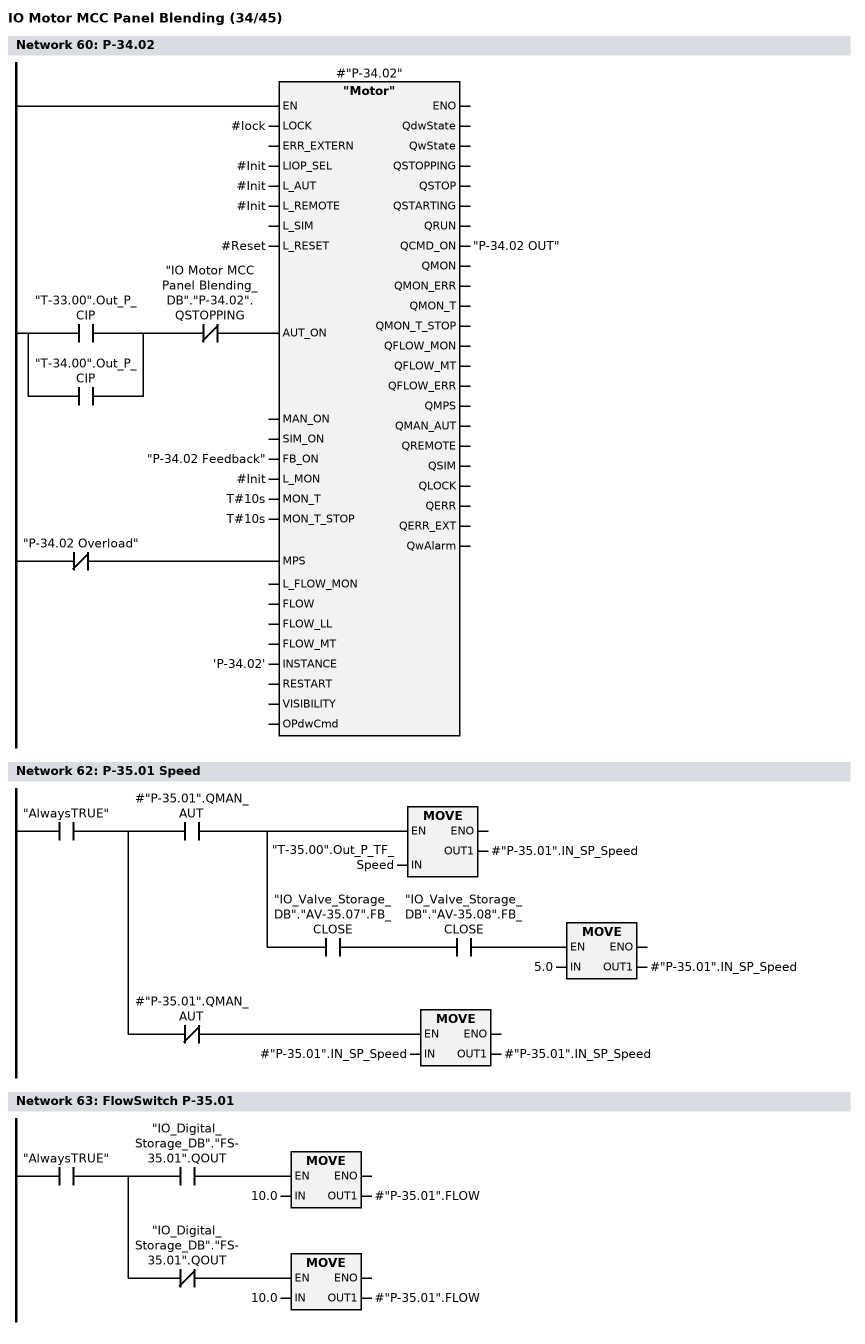
   RUNG wire#powerrail
      #"P-34.02"(AUT_ON := wire#w2, MPS := wire#w3, LOCK := #lock, ERR_EXTERN :=, LIOP_SEL := #Init, L_AUT := #Init, L_REMOTE := #Init, L_SIM :=, L_RESET := #Reset, MAN_ON :=, SIM_ON :=, FB_ON := "P-34.02 Feedback", L_MON := #Init, MON_T := T#10s, MON_T_STOP := T#10s, L_FLOW_MON :=, FLOW :=, FLOW_LL :=, FLOW_MT :=, INSTANCE := 'P-34.02', RESTART :=, VISIBILITY :=, OPdwCmd :=, QdwState =>, QwState =>, QSTOPPING =>, QSTOP =>, QSTARTING =>, QRUN =>, QCMD_ON => "P-34.02 OUT", QMON =>, QMON_ERR =>, QMON_T =>, QMON_T_STOP =>, QFLOW_MON =>, QFLOW_MT =>, QFLOW_ERR =>, QMPS =>, QMAN_AUT =>, QREMOTE =>, QSIM =>, QLOCK =>, QERR =>, QERR_EXT =>, QwAlarm =>)
   END_RUNG
   RUNG wire#powerrail
      Contact( "T-33.00".Out_P_CIP )
      wire#w1
      I_Contact( "IO Motor MCC Panel Blending_DB"."P-34.02".QSTOPPING )
   END_RUNG wire#w2
   RUNG wire#powerrail
      Contact( "T-34.00".Out_P_CIP )
   END_RUNG wire#w1
   RUNG wire#powerrail
      I_Contact( "P-34.02 Overload" )
   END_RUNG wire#w3
   // the same network as SCL:
   #"P-34.02"(LOCK := #lock,   // "Motor"
              LIOP_SEL := #Init,
              L_AUT := #Init,
              L_REMOTE := #Init,
              L_RESET := #Reset,
              AUT_ON := ("T-33.00".Out_P_CIP OR "T-34.00".Out_P_CIP) AND NOT "IO Motor MCC Panel Blending_DB"."P-34.02".QSTOPPING,
              FB_ON := "P-34.02 Feedback",
              L_MON := #Init,
              MON_T := T#10s,
              MON_T_STOP := T#10s,
              MPS := NOT "P-34.02 Overload",
              INSTANCE := 'P-34.02',
              QCMD_ON => "P-34.02 OUT");
END_REGION

REGION Network 62: P-35.01 Speed
   RUNG wire#powerrail
      Contact( "AlwaysTRUE" )
      wire#w1
      Contact( #"P-35.01".QMAN_AUT )
      wire#w2
      Move(in := "T-35.00".Out_P_TF_Speed, out1 => #"P-35.01".IN_SP_Speed)
   END_RUNG
   RUNG wire#w2
      Contact( "IO_Valve_Storage_DB"."AV-35.07".FB_CLOSE )
      Contact( "IO_Valve_Storage_DB"."AV-35.08".FB_CLOSE )
      Move(in := 5.0, out1 => #"P-35.01".IN_SP_Speed)
   END_RUNG
   RUNG wire#w1
      I_Contact( #"P-35.01".QMAN_AUT )
      Move(in := #"P-35.01".IN_SP_Speed, out1 => #"P-35.01".IN_SP_Speed)
   END_RUNG
   // the same network as SCL:
   #_w1 := "AlwaysTRUE" AND #"P-35.01".QMAN_AUT;
   IF #_w1 THEN #"P-35.01".IN_SP_Speed := "T-35.00".Out_P_TF_Speed; END_IF;
   IF #_w1 AND "IO_Valve_Storage_DB"."AV-35.07".FB_CLOSE AND "IO_Valve_Storage_DB"."AV-35.08".FB_CLOSE THEN
       #"P-35.01".IN_SP_Speed := 5.0;
   END_IF;
   IF "AlwaysTRUE" AND NOT #"P-35.01".QMAN_AUT THEN #"P-35.01".IN_SP_Speed := #"P-35.01".IN_SP_Speed; END_IF;
END_REGION

REGION Network 63: FlowSwitch P-35.01
   RUNG wire#powerrail
      Contact( "AlwaysTRUE" )
      wire#w1
      Contact( "IO_Digital_Storage_DB"."FS-35.01".QOUT )
      Move(in := 10.0, out1 => #"P-35.01".FLOW)
   END_RUNG
   RUNG wire#w1
      I_Contact( "IO_Digital_Storage_DB"."FS-35.01".QOUT )
      Move(in := 10.0, out1 => #"P-35.01".FLOW)
   END_RUNG
   // the same network as SCL:
   IF "AlwaysTRUE" AND "IO_Digital_Storage_DB"."FS-35.01".QOUT THEN #"P-35.01".FLOW := 10.0; END_IF;
   IF "AlwaysTRUE" AND NOT "IO_Digital_Storage_DB"."FS-35.01".QOUT THEN #"P-35.01".FLOW := 10.0; END_IF;
END_REGION

REGION Network 64: P-35.01
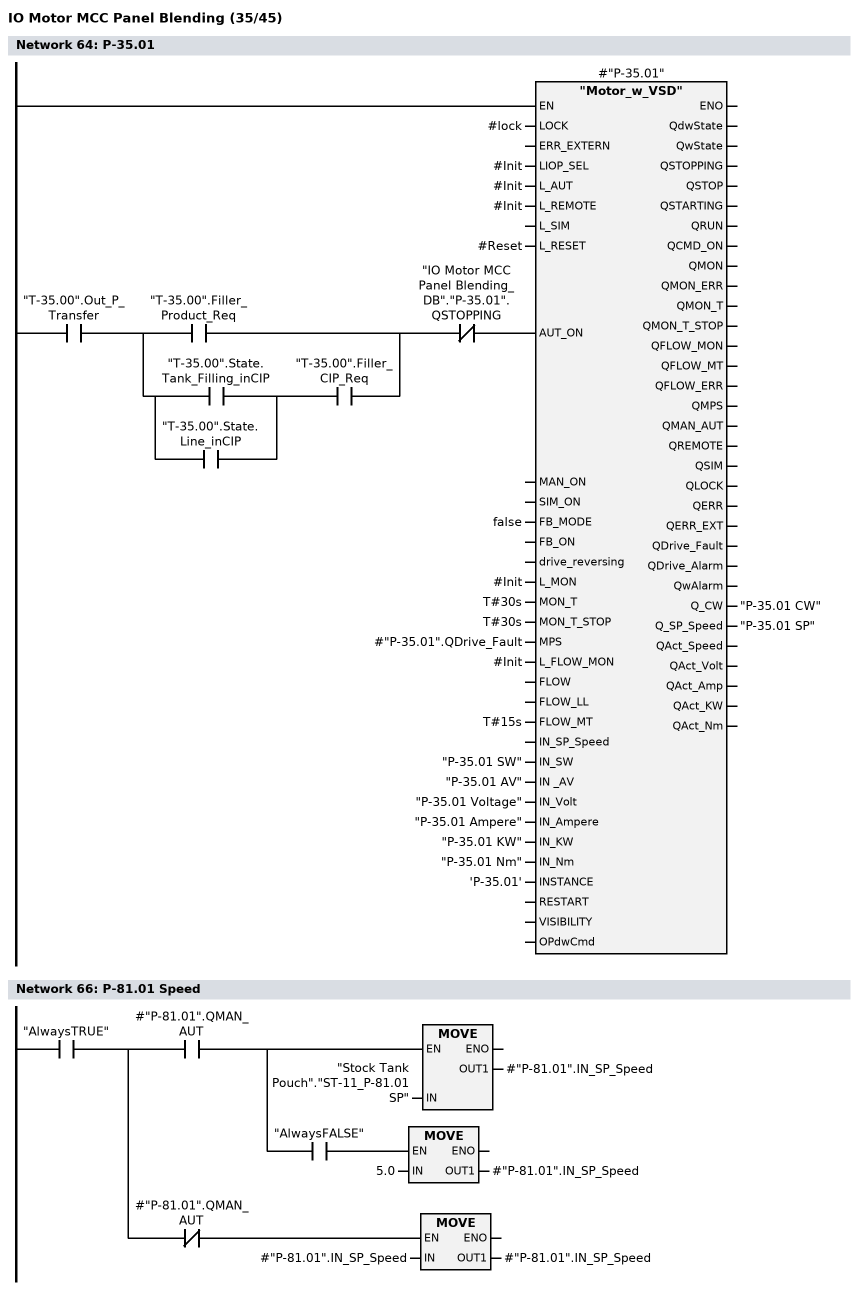
   RUNG wire#powerrail
      #"P-35.01"(AUT_ON := wire#w4, LOCK := #lock, ERR_EXTERN :=, LIOP_SEL := #Init, L_AUT := #Init, L_REMOTE := #Init, L_SIM :=, L_RESET := #Reset, MAN_ON :=, SIM_ON :=, FB_MODE := false, FB_ON :=, drive_reversing :=, L_MON := #Init, MON_T := T#30s, MON_T_STOP := T#30s, MPS := #"P-35.01".QDrive_Fault, L_FLOW_MON := #Init, FLOW :=, FLOW_LL :=, FLOW_MT := T#15s, IN_SP_Speed :=, IN_SW := "P-35.01 SW", "IN _AV" := "P-35.01 AV", IN_Volt := "P-35.01 Voltage", IN_Ampere := "P-35.01 Ampere", IN_KW := "P-35.01 KW", IN_Nm := "P-35.01 Nm", INSTANCE := 'P-35.01', RESTART :=, VISIBILITY :=, OPdwCmd :=, QdwState =>, QwState =>, QSTOPPING =>, QSTOP =>, QSTARTING =>, QRUN =>, QCMD_ON =>, QMON =>, QMON_ERR =>, QMON_T =>, QMON_T_STOP =>, QFLOW_MON =>, QFLOW_MT =>, QFLOW_ERR =>, QMPS =>, QMAN_AUT =>, QREMOTE =>, QSIM =>, QLOCK =>, QERR =>, QERR_EXT =>, QDrive_Fault =>, QDrive_Alarm =>, QwAlarm =>, Q_CW => "P-35.01 CW", Q_SP_Speed => "P-35.01 SP", QAct_Speed =>, QAct_Volt =>, QAct_Amp =>, QAct_KW =>, QAct_Nm =>)
   END_RUNG
   RUNG wire#powerrail
      Contact( "T-35.00".Out_P_Transfer )
      wire#w1
      Contact( "T-35.00".Filler_Product_Req )
      wire#w2
      I_Contact( "IO Motor MCC Panel Blending_DB"."P-35.01".QSTOPPING )
   END_RUNG wire#w4
   RUNG wire#w1
      Contact( "T-35.00".State.Tank_Filling_inCIP )
      wire#w3
      Contact( "T-35.00".Filler_CIP_Req )
   END_RUNG wire#w2
   RUNG wire#w1
      Contact( "T-35.00".State.Line_inCIP )
   END_RUNG wire#w3
   // the same network as SCL:
   #"P-35.01"(LOCK := #lock,   // "Motor_w_VSD"
              LIOP_SEL := #Init,
              L_AUT := #Init,
              L_REMOTE := #Init,
              L_RESET := #Reset,
              AUT_ON := "T-35.00".Out_P_Transfer AND ("T-35.00".Filler_Product_Req OR (("T-35.00".State.Tank_Filling_inCIP OR "T-35.00".State.Line_inCIP) AND "T-35.00".Filler_CIP_Req)) AND NOT "IO Motor MCC Panel Blending_DB"."P-35.01".QSTOPPING,
              FB_MODE := false,
              L_MON := #Init,
              MON_T := T#30s,
              MON_T_STOP := T#30s,
              MPS := #"P-35.01".QDrive_Fault,
              L_FLOW_MON := #Init,
              FLOW_MT := T#15s,
              IN_SW := "P-35.01 SW",
              "IN _AV" := "P-35.01 AV",
              IN_Volt := "P-35.01 Voltage",
              IN_Ampere := "P-35.01 Ampere",
              IN_KW := "P-35.01 KW",
              IN_Nm := "P-35.01 Nm",
              INSTANCE := 'P-35.01',
              Q_CW => "P-35.01 CW",
              Q_SP_Speed => "P-35.01 SP");
END_REGION

REGION Network 66: P-81.01 Speed
   RUNG wire#powerrail
      Contact( "AlwaysTRUE" )
      wire#w1
      Contact( #"P-81.01".QMAN_AUT )
      wire#w2
      Move(in := "Stock Tank Pouch"."ST-11_P-81.01 SP", out1 => #"P-81.01".IN_SP_Speed)
   END_RUNG
   RUNG wire#w2
      Contact( "AlwaysFALSE" )
      Move(in := 5.0, out1 => #"P-81.01".IN_SP_Speed)
   END_RUNG
   RUNG wire#w1
      I_Contact( #"P-81.01".QMAN_AUT )
      Move(in := #"P-81.01".IN_SP_Speed, out1 => #"P-81.01".IN_SP_Speed)
   END_RUNG
   // the same network as SCL:
   #_w1 := "AlwaysTRUE" AND #"P-81.01".QMAN_AUT;
   IF #_w1 THEN #"P-81.01".IN_SP_Speed := "Stock Tank Pouch"."ST-11_P-81.01 SP"; END_IF;
   IF #_w1 AND "AlwaysFALSE" THEN #"P-81.01".IN_SP_Speed := 5.0; END_IF;
   IF "AlwaysTRUE" AND NOT #"P-81.01".QMAN_AUT THEN #"P-81.01".IN_SP_Speed := #"P-81.01".IN_SP_Speed; END_IF;
END_REGION

REGION Network 67: P-81.01
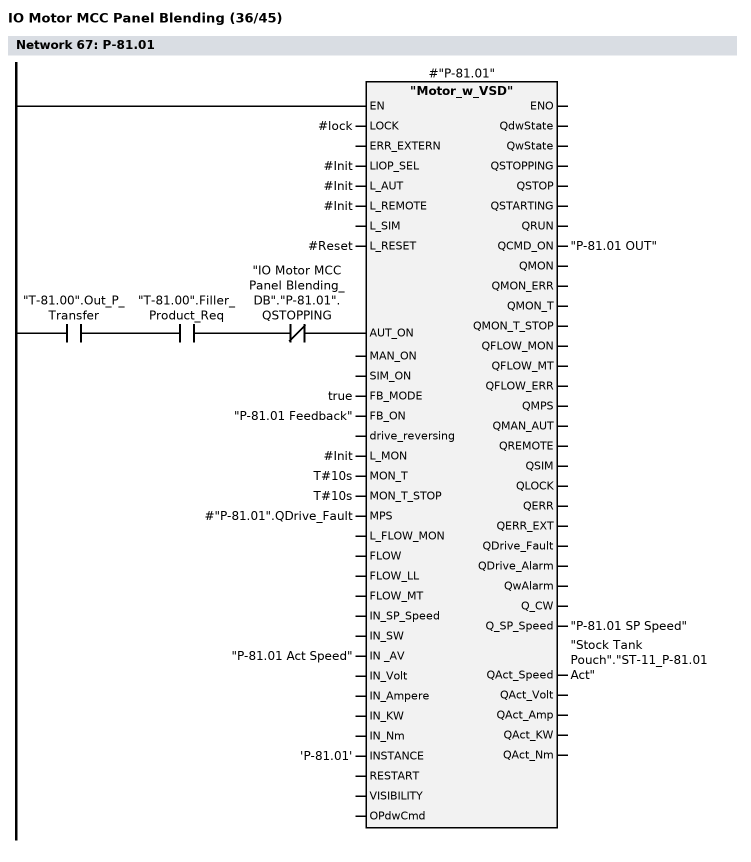
   RUNG wire#powerrail
      #"P-81.01"(AUT_ON := wire#w1, LOCK := #lock, ERR_EXTERN :=, LIOP_SEL := #Init, L_AUT := #Init, L_REMOTE := #Init, L_SIM :=, L_RESET := #Reset, MAN_ON :=, SIM_ON :=, FB_MODE := true, FB_ON := "P-81.01 Feedback", drive_reversing :=, L_MON := #Init, MON_T := T#10s, MON_T_STOP := T#10s, MPS := #"P-81.01".QDrive_Fault, L_FLOW_MON :=, FLOW :=, FLOW_LL :=, FLOW_MT :=, IN_SP_Speed :=, IN_SW :=, "IN _AV" := "P-81.01 Act Speed", IN_Volt :=, IN_Ampere :=, IN_KW :=, IN_Nm :=, INSTANCE := 'P-81.01', RESTART :=, VISIBILITY :=, OPdwCmd :=, QdwState =>, QwState =>, QSTOPPING =>, QSTOP =>, QSTARTING =>, QRUN =>, QCMD_ON => "P-81.01 OUT", QMON =>, QMON_ERR =>, QMON_T =>, QMON_T_STOP =>, QFLOW_MON =>, QFLOW_MT =>, QFLOW_ERR =>, QMPS =>, QMAN_AUT =>, QREMOTE =>, QSIM =>, QLOCK =>, QERR =>, QERR_EXT =>, QDrive_Fault =>, QDrive_Alarm =>, QwAlarm =>, Q_CW =>, Q_SP_Speed => "P-81.01 SP Speed", QAct_Speed => "Stock Tank Pouch"."ST-11_P-81.01 Act", QAct_Volt =>, QAct_Amp =>, QAct_KW =>, QAct_Nm =>)
   END_RUNG
   RUNG wire#powerrail
      Contact( "T-81.00".Out_P_Transfer )
      Contact( "T-81.00".Filler_Product_Req )
      I_Contact( "IO Motor MCC Panel Blending_DB"."P-81.01".QSTOPPING )
   END_RUNG wire#w1
   // the same network as SCL:
   #"P-81.01"(LOCK := #lock,   // "Motor_w_VSD"
              LIOP_SEL := #Init,
              L_AUT := #Init,
              L_REMOTE := #Init,
              L_RESET := #Reset,
              AUT_ON := "T-81.00".Out_P_Transfer AND "T-81.00".Filler_Product_Req AND NOT "IO Motor MCC Panel Blending_DB"."P-81.01".QSTOPPING,
              FB_MODE := true,
              FB_ON := "P-81.01 Feedback",
              L_MON := #Init,
              MON_T := T#10s,
              MON_T_STOP := T#10s,
              MPS := #"P-81.01".QDrive_Fault,
              "IN _AV" := "P-81.01 Act Speed",
              INSTANCE := 'P-81.01',
              QCMD_ON => "P-81.01 OUT",
              Q_SP_Speed => "P-81.01 SP Speed",
              QAct_Speed => "Stock Tank Pouch"."ST-11_P-81.01 Act");
END_REGION

REGION Network 68: P-81.02A
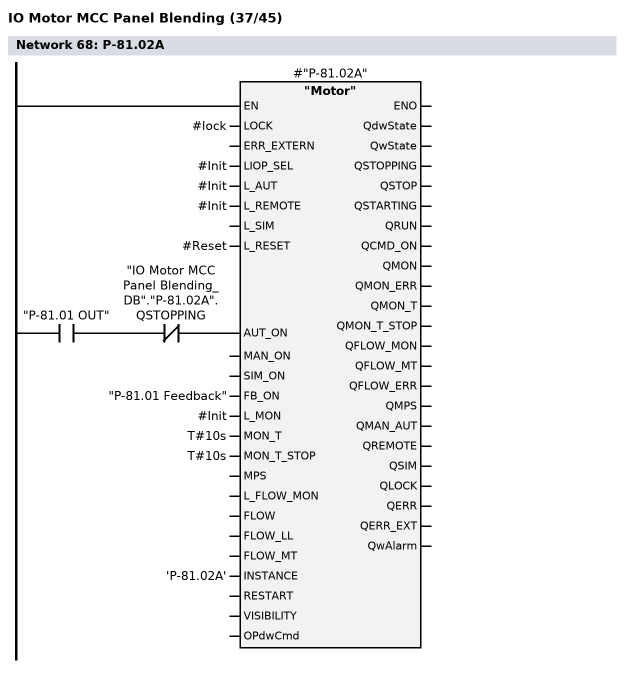
   RUNG wire#powerrail
      #"P-81.02A"(AUT_ON := wire#w1, LOCK := #lock, ERR_EXTERN :=, LIOP_SEL := #Init, L_AUT := #Init, L_REMOTE := #Init, L_SIM :=, L_RESET := #Reset, MAN_ON :=, SIM_ON :=, FB_ON := "P-81.01 Feedback", L_MON := #Init, MON_T := T#10s, MON_T_STOP := T#10s, MPS :=, L_FLOW_MON :=, FLOW :=, FLOW_LL :=, FLOW_MT :=, INSTANCE := 'P-81.02A', RESTART :=, VISIBILITY :=, OPdwCmd :=, QdwState =>, QwState =>, QSTOPPING =>, QSTOP =>, QSTARTING =>, QRUN =>, QCMD_ON =>, QMON =>, QMON_ERR =>, QMON_T =>, QMON_T_STOP =>, QFLOW_MON =>, QFLOW_MT =>, QFLOW_ERR =>, QMPS =>, QMAN_AUT =>, QREMOTE =>, QSIM =>, QLOCK =>, QERR =>, QERR_EXT =>, QwAlarm =>)
   END_RUNG
   RUNG wire#powerrail
      Contact( "P-81.01 OUT" )
      I_Contact( "IO Motor MCC Panel Blending_DB"."P-81.02A".QSTOPPING )
   END_RUNG wire#w1
   // the same network as SCL:
   #"P-81.02A"(LOCK := #lock,   // "Motor"
               LIOP_SEL := #Init,
               L_AUT := #Init,
               L_REMOTE := #Init,
               L_RESET := #Reset,
               AUT_ON := "P-81.01 OUT" AND NOT "IO Motor MCC Panel Blending_DB"."P-81.02A".QSTOPPING,
               FB_ON := "P-81.01 Feedback",
               L_MON := #Init,
               MON_T := T#10s,
               MON_T_STOP := T#10s,
               INSTANCE := 'P-81.02A');
END_REGION

REGION Network 69: P-81.02
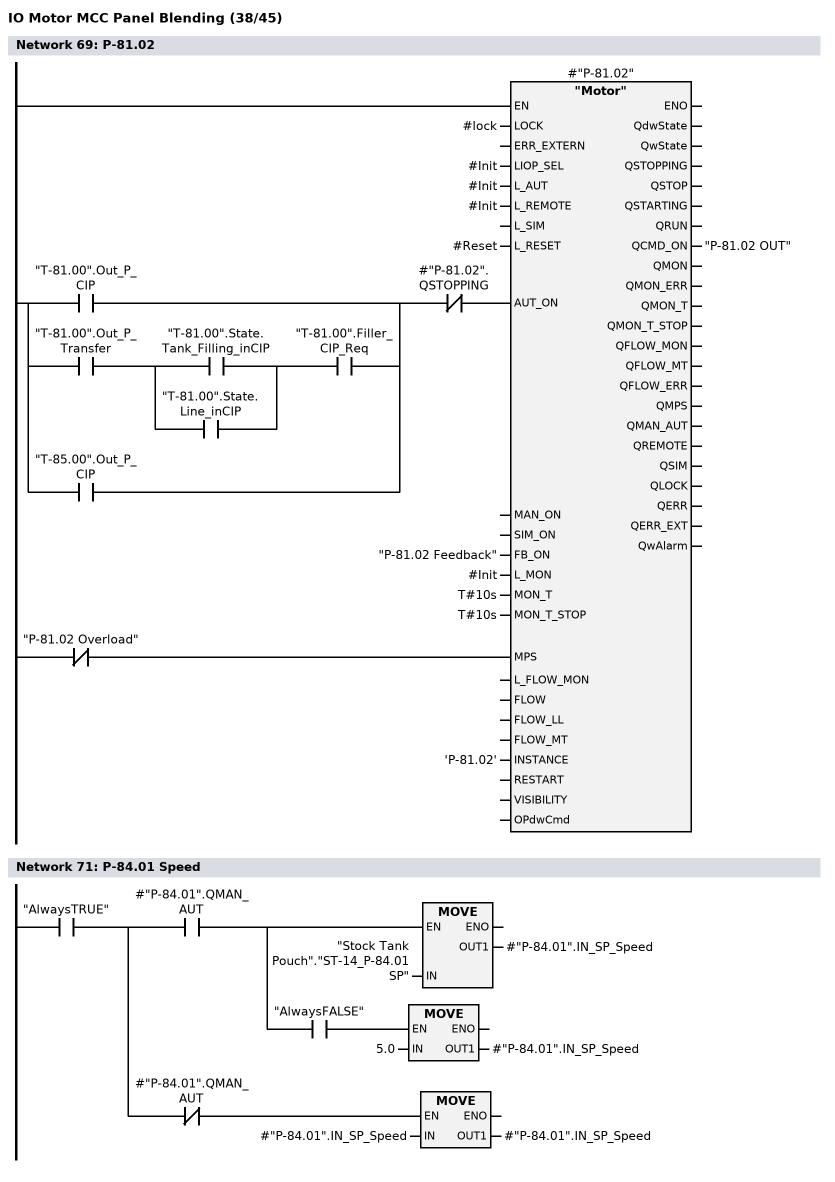
   RUNG wire#powerrail
      #"P-81.02"(AUT_ON := wire#w4, MPS := wire#w5, LOCK := #lock, ERR_EXTERN :=, LIOP_SEL := #Init, L_AUT := #Init, L_REMOTE := #Init, L_SIM :=, L_RESET := #Reset, MAN_ON :=, SIM_ON :=, FB_ON := "P-81.02 Feedback", L_MON := #Init, MON_T := T#10s, MON_T_STOP := T#10s, L_FLOW_MON :=, FLOW :=, FLOW_LL :=, FLOW_MT :=, INSTANCE := 'P-81.02', RESTART :=, VISIBILITY :=, OPdwCmd :=, QdwState =>, QwState =>, QSTOPPING =>, QSTOP =>, QSTARTING =>, QRUN =>, QCMD_ON => "P-81.02 OUT", QMON =>, QMON_ERR =>, QMON_T =>, QMON_T_STOP =>, QFLOW_MON =>, QFLOW_MT =>, QFLOW_ERR =>, QMPS =>, QMAN_AUT =>, QREMOTE =>, QSIM =>, QLOCK =>, QERR =>, QERR_EXT =>, QwAlarm =>)
   END_RUNG
   RUNG wire#powerrail
      Contact( "T-81.00".Out_P_CIP )
      wire#w1
      I_Contact( #"P-81.02".QSTOPPING )
   END_RUNG wire#w4
   RUNG wire#powerrail
      Contact( "T-81.00".Out_P_Transfer )
      wire#w2
      Contact( "T-81.00".State.Tank_Filling_inCIP )
      wire#w3
      Contact( "T-81.00".Filler_CIP_Req )
   END_RUNG wire#w1
   RUNG wire#w2
      Contact( "T-81.00".State.Line_inCIP )
   END_RUNG wire#w3
   RUNG wire#powerrail
      Contact( "T-85.00".Out_P_CIP )
   END_RUNG wire#w1
   RUNG wire#powerrail
      I_Contact( "P-81.02 Overload" )
   END_RUNG wire#w5
   // the same network as SCL:
   #"P-81.02"(LOCK := #lock,   // "Motor"
              LIOP_SEL := #Init,
              L_AUT := #Init,
              L_REMOTE := #Init,
              L_RESET := #Reset,
              AUT_ON := ("T-81.00".Out_P_CIP OR ("T-81.00".Out_P_Transfer AND ("T-81.00".State.Tank_Filling_inCIP OR "T-81.00".State.Line_inCIP) AND "T-81.00".Filler_CIP_Req) OR "T-85.00".Out_P_CIP) AND NOT #"P-81.02".QSTOPPING,
              FB_ON := "P-81.02 Feedback",
              L_MON := #Init,
              MON_T := T#10s,
              MON_T_STOP := T#10s,
              MPS := NOT "P-81.02 Overload",
              INSTANCE := 'P-81.02',
              QCMD_ON => "P-81.02 OUT");
END_REGION

REGION Network 71: P-84.01 Speed
   RUNG wire#powerrail
      Contact( "AlwaysTRUE" )
      wire#w1
      Contact( #"P-84.01".QMAN_AUT )
      wire#w2
      Move(in := "Stock Tank Pouch"."ST-14_P-84.01 SP", out1 => #"P-84.01".IN_SP_Speed)
   END_RUNG
   RUNG wire#w2
      Contact( "AlwaysFALSE" )
      Move(in := 5.0, out1 => #"P-84.01".IN_SP_Speed)
   END_RUNG
   RUNG wire#w1
      I_Contact( #"P-84.01".QMAN_AUT )
      Move(in := #"P-84.01".IN_SP_Speed, out1 => #"P-84.01".IN_SP_Speed)
   END_RUNG
   // the same network as SCL:
   #_w1 := "AlwaysTRUE" AND #"P-84.01".QMAN_AUT;
   IF #_w1 THEN #"P-84.01".IN_SP_Speed := "Stock Tank Pouch"."ST-14_P-84.01 SP"; END_IF;
   IF #_w1 AND "AlwaysFALSE" THEN #"P-84.01".IN_SP_Speed := 5.0; END_IF;
   IF "AlwaysTRUE" AND NOT #"P-84.01".QMAN_AUT THEN #"P-84.01".IN_SP_Speed := #"P-84.01".IN_SP_Speed; END_IF;
END_REGION

REGION Network 72: P-84.01
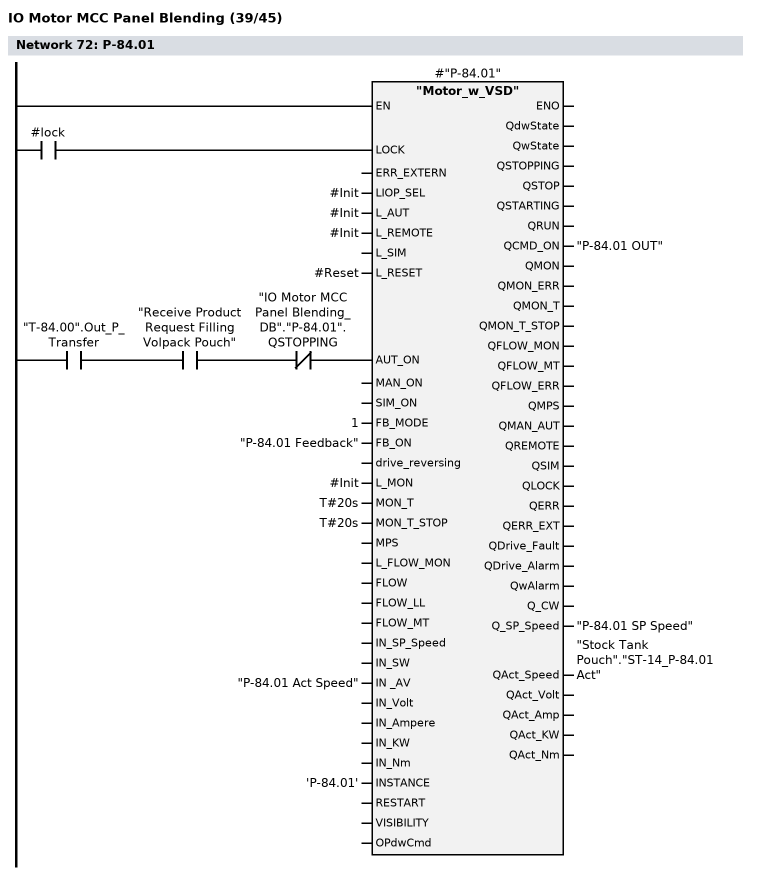
   RUNG wire#powerrail
      #"P-84.01"(LOCK := wire#w1, AUT_ON := wire#w2, ERR_EXTERN :=, LIOP_SEL := #Init, L_AUT := #Init, L_REMOTE := #Init, L_SIM :=, L_RESET := #Reset, MAN_ON :=, SIM_ON :=, FB_MODE := 1, FB_ON := "P-84.01 Feedback", drive_reversing :=, L_MON := #Init, MON_T := T#20s, MON_T_STOP := T#20s, MPS :=, L_FLOW_MON :=, FLOW :=, FLOW_LL :=, FLOW_MT :=, IN_SP_Speed :=, IN_SW :=, "IN _AV" := "P-84.01 Act Speed", IN_Volt :=, IN_Ampere :=, IN_KW :=, IN_Nm :=, INSTANCE := 'P-84.01', RESTART :=, VISIBILITY :=, OPdwCmd :=, QdwState =>, QwState =>, QSTOPPING =>, QSTOP =>, QSTARTING =>, QRUN =>, QCMD_ON => "P-84.01 OUT", QMON =>, QMON_ERR =>, QMON_T =>, QMON_T_STOP =>, QFLOW_MON =>, QFLOW_MT =>, QFLOW_ERR =>, QMPS =>, QMAN_AUT =>, QREMOTE =>, QSIM =>, QLOCK =>, QERR =>, QERR_EXT =>, QDrive_Fault =>, QDrive_Alarm =>, QwAlarm =>, Q_CW =>, Q_SP_Speed => "P-84.01 SP Speed", QAct_Speed => "Stock Tank Pouch"."ST-14_P-84.01 Act", QAct_Volt =>, QAct_Amp =>, QAct_KW =>, QAct_Nm =>)
   END_RUNG
   RUNG wire#powerrail
      Contact( #lock )
   END_RUNG wire#w1
   RUNG wire#powerrail
      Contact( "T-84.00".Out_P_Transfer )
      Contact( "Receive Product Request Filling Volpack Pouch" )
      I_Contact( "IO Motor MCC Panel Blending_DB"."P-84.01".QSTOPPING )
   END_RUNG wire#w2
   // the same network as SCL:
   #"P-84.01"(LOCK := #lock,   // "Motor_w_VSD"
              LIOP_SEL := #Init,
              L_AUT := #Init,
              L_REMOTE := #Init,
              L_RESET := #Reset,
              AUT_ON := "T-84.00".Out_P_Transfer AND "Receive Product Request Filling Volpack Pouch" AND NOT "IO Motor MCC Panel Blending_DB"."P-84.01".QSTOPPING,
              FB_MODE := 1,
              FB_ON := "P-84.01 Feedback",
              L_MON := #Init,
              MON_T := T#20s,
              MON_T_STOP := T#20s,
              "IN _AV" := "P-84.01 Act Speed",
              INSTANCE := 'P-84.01',
              QCMD_ON => "P-84.01 OUT",
              Q_SP_Speed => "P-84.01 SP Speed",
              QAct_Speed => "Stock Tank Pouch"."ST-14_P-84.01 Act");
END_REGION

REGION Network 73: P-84.01A
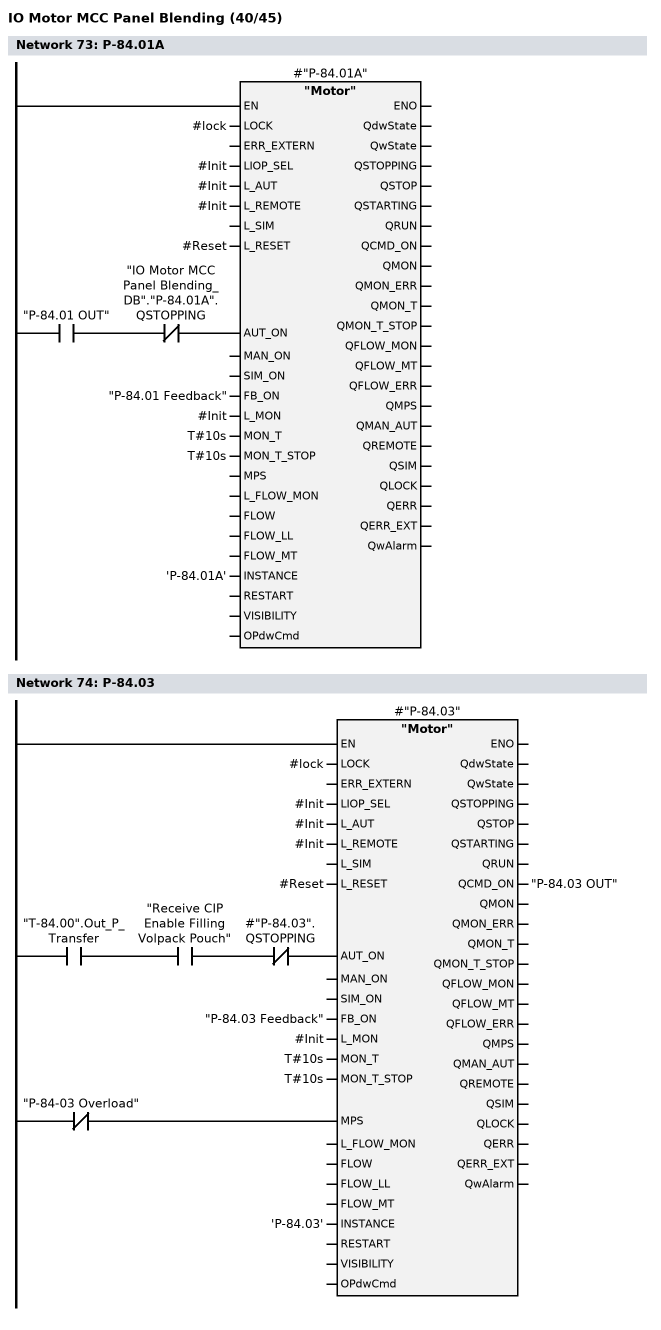
   RUNG wire#powerrail
      #"P-84.01A"(AUT_ON := wire#w1, LOCK := #lock, ERR_EXTERN :=, LIOP_SEL := #Init, L_AUT := #Init, L_REMOTE := #Init, L_SIM :=, L_RESET := #Reset, MAN_ON :=, SIM_ON :=, FB_ON := "P-84.01 Feedback", L_MON := #Init, MON_T := T#10s, MON_T_STOP := T#10s, MPS :=, L_FLOW_MON :=, FLOW :=, FLOW_LL :=, FLOW_MT :=, INSTANCE := 'P-84.01A', RESTART :=, VISIBILITY :=, OPdwCmd :=, QdwState =>, QwState =>, QSTOPPING =>, QSTOP =>, QSTARTING =>, QRUN =>, QCMD_ON =>, QMON =>, QMON_ERR =>, QMON_T =>, QMON_T_STOP =>, QFLOW_MON =>, QFLOW_MT =>, QFLOW_ERR =>, QMPS =>, QMAN_AUT =>, QREMOTE =>, QSIM =>, QLOCK =>, QERR =>, QERR_EXT =>, QwAlarm =>)
   END_RUNG
   RUNG wire#powerrail
      Contact( "P-84.01 OUT" )
      I_Contact( "IO Motor MCC Panel Blending_DB"."P-84.01A".QSTOPPING )
   END_RUNG wire#w1
   // the same network as SCL:
   #"P-84.01A"(LOCK := #lock,   // "Motor"
               LIOP_SEL := #Init,
               L_AUT := #Init,
               L_REMOTE := #Init,
               L_RESET := #Reset,
               AUT_ON := "P-84.01 OUT" AND NOT "IO Motor MCC Panel Blending_DB"."P-84.01A".QSTOPPING,
               FB_ON := "P-84.01 Feedback",
               L_MON := #Init,
               MON_T := T#10s,
               MON_T_STOP := T#10s,
               INSTANCE := 'P-84.01A');
END_REGION

REGION Network 74: P-84.03
   RUNG wire#powerrail
      #"P-84.03"(AUT_ON := wire#w1, MPS := wire#w2, LOCK := #lock, ERR_EXTERN :=, LIOP_SEL := #Init, L_AUT := #Init, L_REMOTE := #Init, L_SIM :=, L_RESET := #Reset, MAN_ON :=, SIM_ON :=, FB_ON := "P-84.03 Feedback", L_MON := #Init, MON_T := T#10s, MON_T_STOP := T#10s, L_FLOW_MON :=, FLOW :=, FLOW_LL :=, FLOW_MT :=, INSTANCE := 'P-84.03', RESTART :=, VISIBILITY :=, OPdwCmd :=, QdwState =>, QwState =>, QSTOPPING =>, QSTOP =>, QSTARTING =>, QRUN =>, QCMD_ON => "P-84.03 OUT", QMON =>, QMON_ERR =>, QMON_T =>, QMON_T_STOP =>, QFLOW_MON =>, QFLOW_MT =>, QFLOW_ERR =>, QMPS =>, QMAN_AUT =>, QREMOTE =>, QSIM =>, QLOCK =>, QERR =>, QERR_EXT =>, QwAlarm =>)
   END_RUNG
   RUNG wire#powerrail
      Contact( "T-84.00".Out_P_Transfer )
      Contact( "Receive CIP Enable Filling Volpack Pouch" )
      I_Contact( #"P-84.03".QSTOPPING )
   END_RUNG wire#w1
   RUNG wire#powerrail
      I_Contact( "P-84-03 Overload" )
   END_RUNG wire#w2
   // the same network as SCL:
   #"P-84.03"(LOCK := #lock,   // "Motor"
              LIOP_SEL := #Init,
              L_AUT := #Init,
              L_REMOTE := #Init,
              L_RESET := #Reset,
              AUT_ON := "T-84.00".Out_P_Transfer AND "Receive CIP Enable Filling Volpack Pouch" AND NOT #"P-84.03".QSTOPPING,
              FB_ON := "P-84.03 Feedback",
              L_MON := #Init,
              MON_T := T#10s,
              MON_T_STOP := T#10s,
              MPS := NOT "P-84-03 Overload",
              INSTANCE := 'P-84.03',
              QCMD_ON => "P-84.03 OUT");
END_REGION

REGION Network 75: P-84.02 Speed
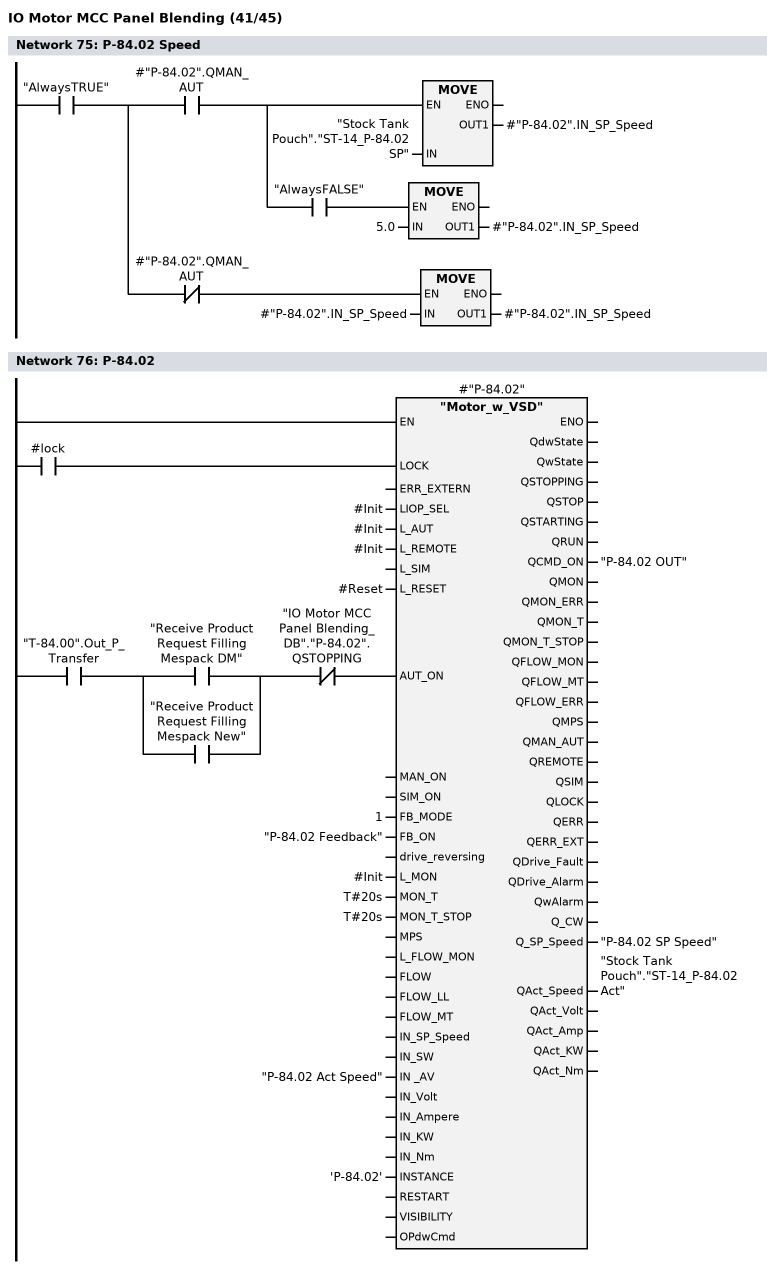
   RUNG wire#powerrail
      Contact( "AlwaysTRUE" )
      wire#w1
      Contact( #"P-84.02".QMAN_AUT )
      wire#w2
      Move(in := "Stock Tank Pouch"."ST-14_P-84.02 SP", out1 => #"P-84.02".IN_SP_Speed)
   END_RUNG
   RUNG wire#w2
      Contact( "AlwaysFALSE" )
      Move(in := 5.0, out1 => #"P-84.02".IN_SP_Speed)
   END_RUNG
   RUNG wire#w1
      I_Contact( #"P-84.02".QMAN_AUT )
      Move(in := #"P-84.02".IN_SP_Speed, out1 => #"P-84.02".IN_SP_Speed)
   END_RUNG
   // the same network as SCL:
   #_w1 := "AlwaysTRUE" AND #"P-84.02".QMAN_AUT;
   IF #_w1 THEN #"P-84.02".IN_SP_Speed := "Stock Tank Pouch"."ST-14_P-84.02 SP"; END_IF;
   IF #_w1 AND "AlwaysFALSE" THEN #"P-84.02".IN_SP_Speed := 5.0; END_IF;
   IF "AlwaysTRUE" AND NOT #"P-84.02".QMAN_AUT THEN #"P-84.02".IN_SP_Speed := #"P-84.02".IN_SP_Speed; END_IF;
END_REGION

REGION Network 76: P-84.02
   RUNG wire#powerrail
      #"P-84.02"(LOCK := wire#w1, AUT_ON := wire#w4, ERR_EXTERN :=, LIOP_SEL := #Init, L_AUT := #Init, L_REMOTE := #Init, L_SIM :=, L_RESET := #Reset, MAN_ON :=, SIM_ON :=, FB_MODE := 1, FB_ON := "P-84.02 Feedback", drive_reversing :=, L_MON := #Init, MON_T := T#20s, MON_T_STOP := T#20s, MPS :=, L_FLOW_MON :=, FLOW :=, FLOW_LL :=, FLOW_MT :=, IN_SP_Speed :=, IN_SW :=, "IN _AV" := "P-84.02 Act Speed", IN_Volt :=, IN_Ampere :=, IN_KW :=, IN_Nm :=, INSTANCE := 'P-84.02', RESTART :=, VISIBILITY :=, OPdwCmd :=, QdwState =>, QwState =>, QSTOPPING =>, QSTOP =>, QSTARTING =>, QRUN =>, QCMD_ON => "P-84.02 OUT", QMON =>, QMON_ERR =>, QMON_T =>, QMON_T_STOP =>, QFLOW_MON =>, QFLOW_MT =>, QFLOW_ERR =>, QMPS =>, QMAN_AUT =>, QREMOTE =>, QSIM =>, QLOCK =>, QERR =>, QERR_EXT =>, QDrive_Fault =>, QDrive_Alarm =>, QwAlarm =>, Q_CW =>, Q_SP_Speed => "P-84.02 SP Speed", QAct_Speed => "Stock Tank Pouch"."ST-14_P-84.02 Act", QAct_Volt =>, QAct_Amp =>, QAct_KW =>, QAct_Nm =>)
   END_RUNG
   RUNG wire#powerrail
      Contact( #lock )
   END_RUNG wire#w1
   RUNG wire#powerrail
      Contact( "T-84.00".Out_P_Transfer )
      wire#w2
      Contact( "Receive Product Request Filling Mespack DM" )
      wire#w3
      I_Contact( "IO Motor MCC Panel Blending_DB"."P-84.02".QSTOPPING )
   END_RUNG wire#w4
   RUNG wire#w2
      Contact( "Receive Product Request Filling Mespack New" )
   END_RUNG wire#w3
   // the same network as SCL:
   #"P-84.02"(LOCK := #lock,   // "Motor_w_VSD"
              LIOP_SEL := #Init,
              L_AUT := #Init,
              L_REMOTE := #Init,
              L_RESET := #Reset,
              AUT_ON := "T-84.00".Out_P_Transfer AND ("Receive Product Request Filling Mespack DM" OR "Receive Product Request Filling Mespack New") AND NOT "IO Motor MCC Panel Blending_DB"."P-84.02".QSTOPPING,
              FB_MODE := 1,
              FB_ON := "P-84.02 Feedback",
              L_MON := #Init,
              MON_T := T#20s,
              MON_T_STOP := T#20s,
              "IN _AV" := "P-84.02 Act Speed",
              INSTANCE := 'P-84.02',
              QCMD_ON => "P-84.02 OUT",
              Q_SP_Speed => "P-84.02 SP Speed",
              QAct_Speed => "Stock Tank Pouch"."ST-14_P-84.02 Act");
END_REGION

REGION Network 77: P-84.02A
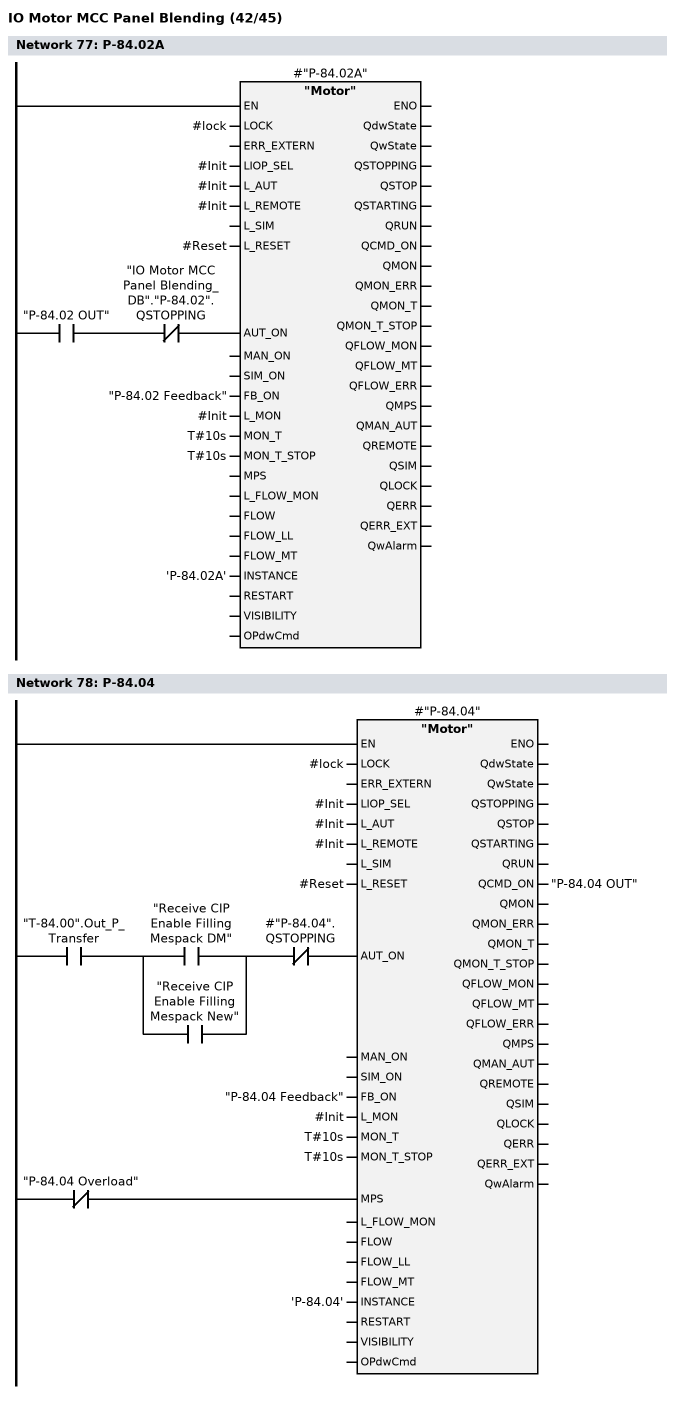
   RUNG wire#powerrail
      #"P-84.02A"(AUT_ON := wire#w1, LOCK := #lock, ERR_EXTERN :=, LIOP_SEL := #Init, L_AUT := #Init, L_REMOTE := #Init, L_SIM :=, L_RESET := #Reset, MAN_ON :=, SIM_ON :=, FB_ON := "P-84.02 Feedback", L_MON := #Init, MON_T := T#10s, MON_T_STOP := T#10s, MPS :=, L_FLOW_MON :=, FLOW :=, FLOW_LL :=, FLOW_MT :=, INSTANCE := 'P-84.02A', RESTART :=, VISIBILITY :=, OPdwCmd :=, QdwState =>, QwState =>, QSTOPPING =>, QSTOP =>, QSTARTING =>, QRUN =>, QCMD_ON =>, QMON =>, QMON_ERR =>, QMON_T =>, QMON_T_STOP =>, QFLOW_MON =>, QFLOW_MT =>, QFLOW_ERR =>, QMPS =>, QMAN_AUT =>, QREMOTE =>, QSIM =>, QLOCK =>, QERR =>, QERR_EXT =>, QwAlarm =>)
   END_RUNG
   RUNG wire#powerrail
      Contact( "P-84.02 OUT" )
      I_Contact( "IO Motor MCC Panel Blending_DB"."P-84.02".QSTOPPING )
   END_RUNG wire#w1
   // the same network as SCL:
   #"P-84.02A"(LOCK := #lock,   // "Motor"
               LIOP_SEL := #Init,
               L_AUT := #Init,
               L_REMOTE := #Init,
               L_RESET := #Reset,
               AUT_ON := "P-84.02 OUT" AND NOT "IO Motor MCC Panel Blending_DB"."P-84.02".QSTOPPING,
               FB_ON := "P-84.02 Feedback",
               L_MON := #Init,
               MON_T := T#10s,
               MON_T_STOP := T#10s,
               INSTANCE := 'P-84.02A');
END_REGION

REGION Network 78: P-84.04
   RUNG wire#powerrail
      #"P-84.04"(AUT_ON := wire#w3, MPS := wire#w4, LOCK := #lock, ERR_EXTERN :=, LIOP_SEL := #Init, L_AUT := #Init, L_REMOTE := #Init, L_SIM :=, L_RESET := #Reset, MAN_ON :=, SIM_ON :=, FB_ON := "P-84.04 Feedback", L_MON := #Init, MON_T := T#10s, MON_T_STOP := T#10s, L_FLOW_MON :=, FLOW :=, FLOW_LL :=, FLOW_MT :=, INSTANCE := 'P-84.04', RESTART :=, VISIBILITY :=, OPdwCmd :=, QdwState =>, QwState =>, QSTOPPING =>, QSTOP =>, QSTARTING =>, QRUN =>, QCMD_ON => "P-84.04 OUT", QMON =>, QMON_ERR =>, QMON_T =>, QMON_T_STOP =>, QFLOW_MON =>, QFLOW_MT =>, QFLOW_ERR =>, QMPS =>, QMAN_AUT =>, QREMOTE =>, QSIM =>, QLOCK =>, QERR =>, QERR_EXT =>, QwAlarm =>)
   END_RUNG
   RUNG wire#powerrail
      Contact( "T-84.00".Out_P_Transfer )
      wire#w1
      Contact( "Receive CIP Enable Filling Mespack DM" )
      wire#w2
      I_Contact( #"P-84.04".QSTOPPING )
   END_RUNG wire#w3
   RUNG wire#w1
      Contact( "Receive CIP Enable Filling Mespack New" )
   END_RUNG wire#w2
   RUNG wire#powerrail
      I_Contact( "P-84.04 Overload" )
   END_RUNG wire#w4
   // the same network as SCL:
   #"P-84.04"(LOCK := #lock,   // "Motor"
              LIOP_SEL := #Init,
              L_AUT := #Init,
              L_REMOTE := #Init,
              L_RESET := #Reset,
              AUT_ON := "T-84.00".Out_P_Transfer AND ("Receive CIP Enable Filling Mespack DM" OR "Receive CIP Enable Filling Mespack New") AND NOT #"P-84.04".QSTOPPING,
              FB_ON := "P-84.04 Feedback",
              L_MON := #Init,
              MON_T := T#10s,
              MON_T_STOP := T#10s,
              MPS := NOT "P-84.04 Overload",
              INSTANCE := 'P-84.04',
              QCMD_ON => "P-84.04 OUT");
END_REGION

REGION Network 80: P-82.01 Speed
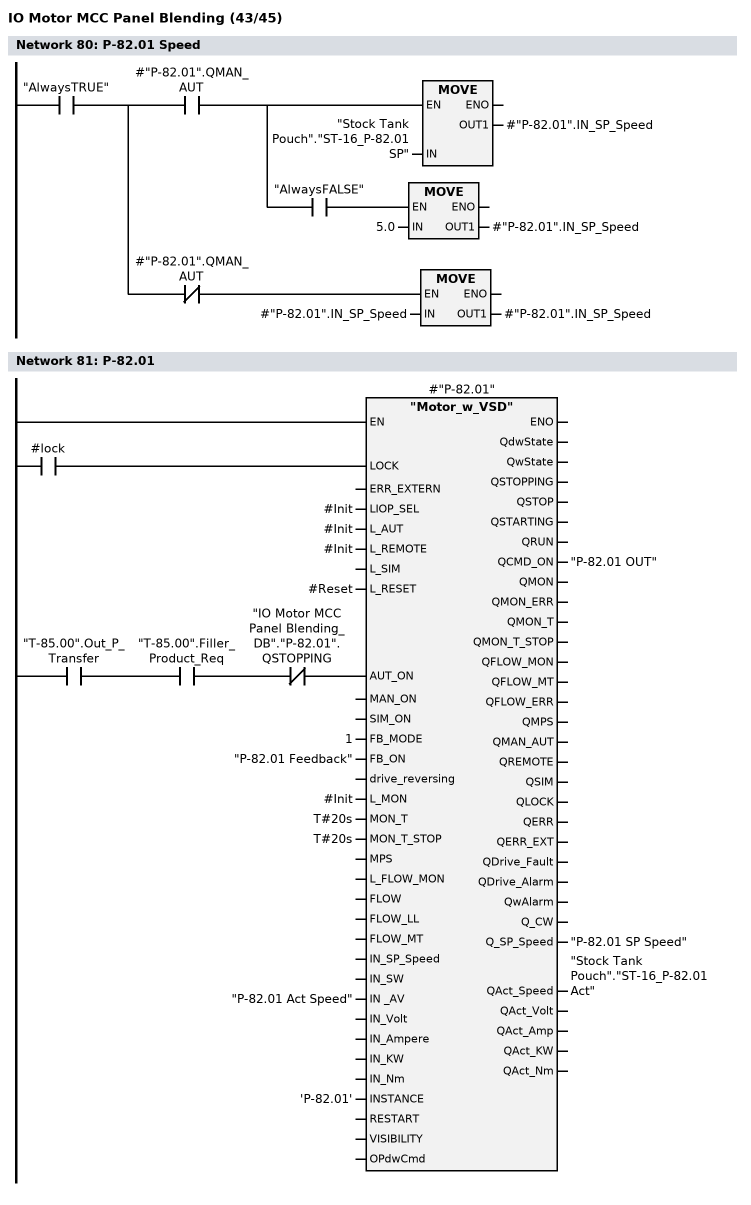
   RUNG wire#powerrail
      Contact( "AlwaysTRUE" )
      wire#w1
      Contact( #"P-82.01".QMAN_AUT )
      wire#w2
      Move(in := "Stock Tank Pouch"."ST-16_P-82.01 SP", out1 => #"P-82.01".IN_SP_Speed)
   END_RUNG
   RUNG wire#w2
      Contact( "AlwaysFALSE" )
      Move(in := 5.0, out1 => #"P-82.01".IN_SP_Speed)
   END_RUNG
   RUNG wire#w1
      I_Contact( #"P-82.01".QMAN_AUT )
      Move(in := #"P-82.01".IN_SP_Speed, out1 => #"P-82.01".IN_SP_Speed)
   END_RUNG
   // the same network as SCL:
   #_w1 := "AlwaysTRUE" AND #"P-82.01".QMAN_AUT;
   IF #_w1 THEN #"P-82.01".IN_SP_Speed := "Stock Tank Pouch"."ST-16_P-82.01 SP"; END_IF;
   IF #_w1 AND "AlwaysFALSE" THEN #"P-82.01".IN_SP_Speed := 5.0; END_IF;
   IF "AlwaysTRUE" AND NOT #"P-82.01".QMAN_AUT THEN #"P-82.01".IN_SP_Speed := #"P-82.01".IN_SP_Speed; END_IF;
END_REGION

REGION Network 81: P-82.01
   RUNG wire#powerrail
      #"P-82.01"(LOCK := wire#w1, AUT_ON := wire#w2, ERR_EXTERN :=, LIOP_SEL := #Init, L_AUT := #Init, L_REMOTE := #Init, L_SIM :=, L_RESET := #Reset, MAN_ON :=, SIM_ON :=, FB_MODE := 1, FB_ON := "P-82.01 Feedback", drive_reversing :=, L_MON := #Init, MON_T := T#20s, MON_T_STOP := T#20s, MPS :=, L_FLOW_MON :=, FLOW :=, FLOW_LL :=, FLOW_MT :=, IN_SP_Speed :=, IN_SW :=, "IN _AV" := "P-82.01 Act Speed", IN_Volt :=, IN_Ampere :=, IN_KW :=, IN_Nm :=, INSTANCE := 'P-82.01', RESTART :=, VISIBILITY :=, OPdwCmd :=, QdwState =>, QwState =>, QSTOPPING =>, QSTOP =>, QSTARTING =>, QRUN =>, QCMD_ON => "P-82.01 OUT", QMON =>, QMON_ERR =>, QMON_T =>, QMON_T_STOP =>, QFLOW_MON =>, QFLOW_MT =>, QFLOW_ERR =>, QMPS =>, QMAN_AUT =>, QREMOTE =>, QSIM =>, QLOCK =>, QERR =>, QERR_EXT =>, QDrive_Fault =>, QDrive_Alarm =>, QwAlarm =>, Q_CW =>, Q_SP_Speed => "P-82.01 SP Speed", QAct_Speed => "Stock Tank Pouch"."ST-16_P-82.01 Act", QAct_Volt =>, QAct_Amp =>, QAct_KW =>, QAct_Nm =>)
   END_RUNG
   RUNG wire#powerrail
      Contact( #lock )
   END_RUNG wire#w1
   RUNG wire#powerrail
      Contact( "T-85.00".Out_P_Transfer )
      Contact( "T-85.00".Filler_Product_Req )
      I_Contact( "IO Motor MCC Panel Blending_DB"."P-82.01".QSTOPPING )
   END_RUNG wire#w2
   // the same network as SCL:
   #"P-82.01"(LOCK := #lock,   // "Motor_w_VSD"
              LIOP_SEL := #Init,
              L_AUT := #Init,
              L_REMOTE := #Init,
              L_RESET := #Reset,
              AUT_ON := "T-85.00".Out_P_Transfer AND "T-85.00".Filler_Product_Req AND NOT "IO Motor MCC Panel Blending_DB"."P-82.01".QSTOPPING,
              FB_MODE := 1,
              FB_ON := "P-82.01 Feedback",
              L_MON := #Init,
              MON_T := T#20s,
              MON_T_STOP := T#20s,
              "IN _AV" := "P-82.01 Act Speed",
              INSTANCE := 'P-82.01',
              QCMD_ON => "P-82.01 OUT",
              Q_SP_Speed => "P-82.01 SP Speed",
              QAct_Speed => "Stock Tank Pouch"."ST-16_P-82.01 Act");
END_REGION

REGION Network 82: P-82.01A
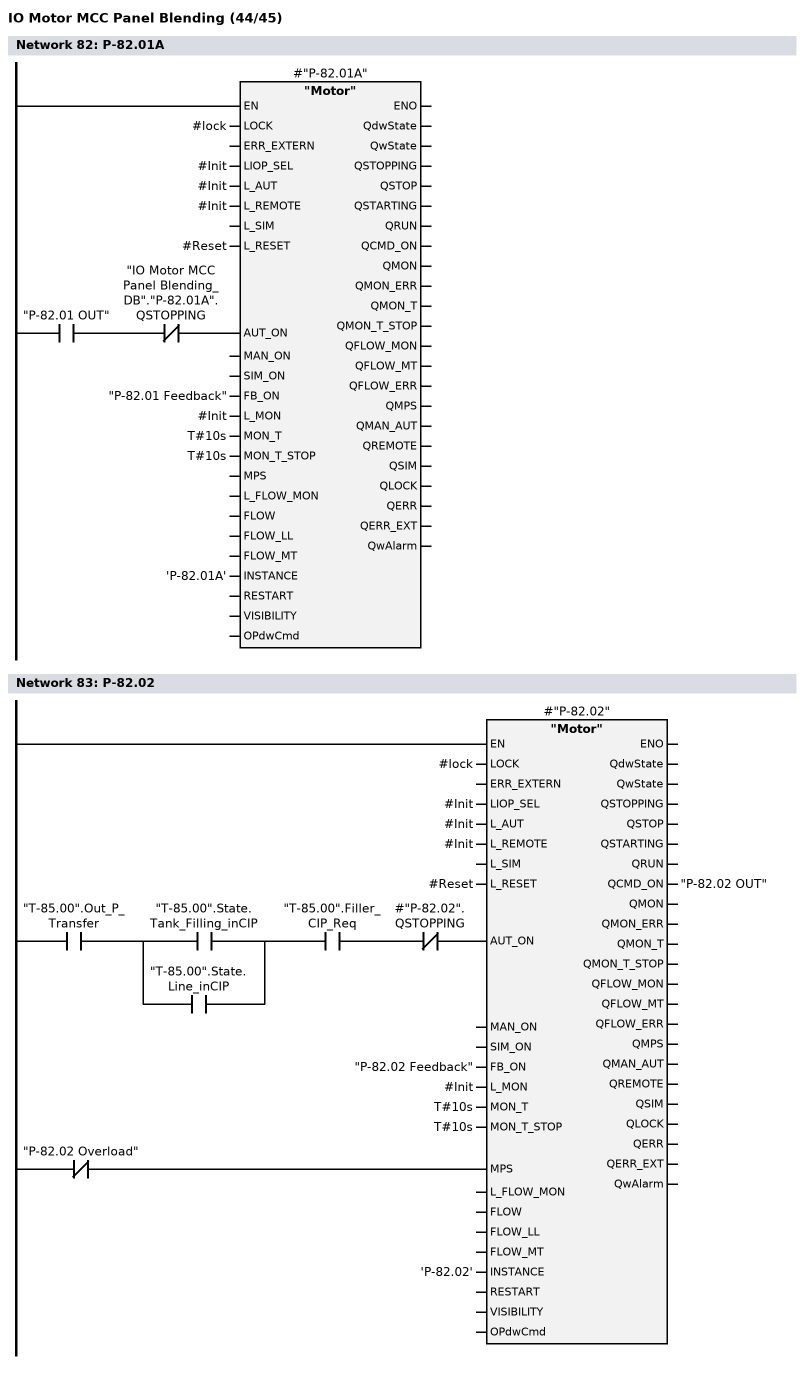
   RUNG wire#powerrail
      #"P-82.01A"(AUT_ON := wire#w1, LOCK := #lock, ERR_EXTERN :=, LIOP_SEL := #Init, L_AUT := #Init, L_REMOTE := #Init, L_SIM :=, L_RESET := #Reset, MAN_ON :=, SIM_ON :=, FB_ON := "P-82.01 Feedback", L_MON := #Init, MON_T := T#10s, MON_T_STOP := T#10s, MPS :=, L_FLOW_MON :=, FLOW :=, FLOW_LL :=, FLOW_MT :=, INSTANCE := 'P-82.01A', RESTART :=, VISIBILITY :=, OPdwCmd :=, QdwState =>, QwState =>, QSTOPPING =>, QSTOP =>, QSTARTING =>, QRUN =>, QCMD_ON =>, QMON =>, QMON_ERR =>, QMON_T =>, QMON_T_STOP =>, QFLOW_MON =>, QFLOW_MT =>, QFLOW_ERR =>, QMPS =>, QMAN_AUT =>, QREMOTE =>, QSIM =>, QLOCK =>, QERR =>, QERR_EXT =>, QwAlarm =>)
   END_RUNG
   RUNG wire#powerrail
      Contact( "P-82.01 OUT" )
      I_Contact( "IO Motor MCC Panel Blending_DB"."P-82.01A".QSTOPPING )
   END_RUNG wire#w1
   // the same network as SCL:
   #"P-82.01A"(LOCK := #lock,   // "Motor"
               LIOP_SEL := #Init,
               L_AUT := #Init,
               L_REMOTE := #Init,
               L_RESET := #Reset,
               AUT_ON := "P-82.01 OUT" AND NOT "IO Motor MCC Panel Blending_DB"."P-82.01A".QSTOPPING,
               FB_ON := "P-82.01 Feedback",
               L_MON := #Init,
               MON_T := T#10s,
               MON_T_STOP := T#10s,
               INSTANCE := 'P-82.01A');
END_REGION

REGION Network 83: P-82.02
   RUNG wire#powerrail
      #"P-82.02"(AUT_ON := wire#w3, MPS := wire#w4, LOCK := #lock, ERR_EXTERN :=, LIOP_SEL := #Init, L_AUT := #Init, L_REMOTE := #Init, L_SIM :=, L_RESET := #Reset, MAN_ON :=, SIM_ON :=, FB_ON := "P-82.02 Feedback", L_MON := #Init, MON_T := T#10s, MON_T_STOP := T#10s, L_FLOW_MON :=, FLOW :=, FLOW_LL :=, FLOW_MT :=, INSTANCE := 'P-82.02', RESTART :=, VISIBILITY :=, OPdwCmd :=, QdwState =>, QwState =>, QSTOPPING =>, QSTOP =>, QSTARTING =>, QRUN =>, QCMD_ON => "P-82.02 OUT", QMON =>, QMON_ERR =>, QMON_T =>, QMON_T_STOP =>, QFLOW_MON =>, QFLOW_MT =>, QFLOW_ERR =>, QMPS =>, QMAN_AUT =>, QREMOTE =>, QSIM =>, QLOCK =>, QERR =>, QERR_EXT =>, QwAlarm =>)
   END_RUNG
   RUNG wire#powerrail
      Contact( "T-85.00".Out_P_Transfer )
      wire#w1
      Contact( "T-85.00".State.Tank_Filling_inCIP )
      wire#w2
      Contact( "T-85.00".Filler_CIP_Req )
      I_Contact( #"P-82.02".QSTOPPING )
   END_RUNG wire#w3
   RUNG wire#w1
      Contact( "T-85.00".State.Line_inCIP )
   END_RUNG wire#w2
   RUNG wire#powerrail
      I_Contact( "P-82.02 Overload" )
   END_RUNG wire#w4
   // the same network as SCL:
   #"P-82.02"(LOCK := #lock,   // "Motor"
              LIOP_SEL := #Init,
              L_AUT := #Init,
              L_REMOTE := #Init,
              L_RESET := #Reset,
              AUT_ON := "T-85.00".Out_P_Transfer AND ("T-85.00".State.Tank_Filling_inCIP OR "T-85.00".State.Line_inCIP) AND "T-85.00".Filler_CIP_Req AND NOT #"P-82.02".QSTOPPING,
              FB_ON := "P-82.02 Feedback",
              L_MON := #Init,
              MON_T := T#10s,
              MON_T_STOP := T#10s,
              MPS := NOT "P-82.02 Overload",
              INSTANCE := 'P-82.02',
              QCMD_ON => "P-82.02 OUT");
END_REGION

REGION Network 84: XA-82.00
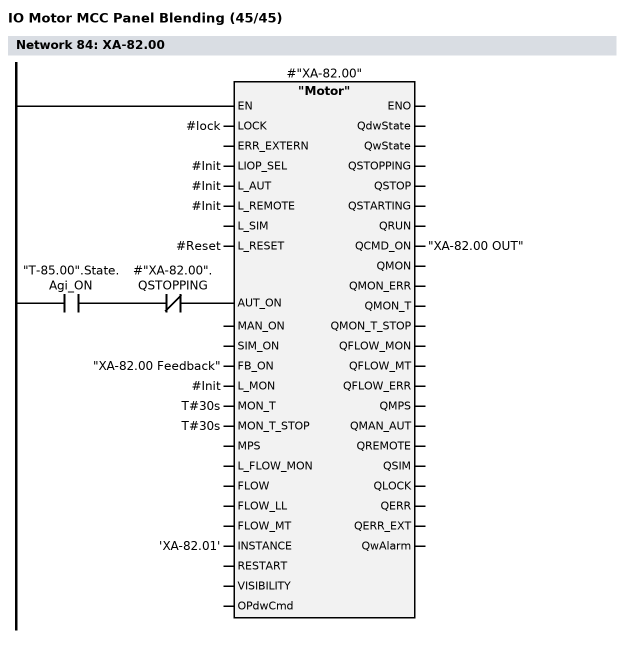
   RUNG wire#powerrail
      #"XA-82.00"(AUT_ON := wire#w1, LOCK := #lock, ERR_EXTERN :=, LIOP_SEL := #Init, L_AUT := #Init, L_REMOTE := #Init, L_SIM :=, L_RESET := #Reset, MAN_ON :=, SIM_ON :=, FB_ON := "XA-82.00 Feedback", L_MON := #Init, MON_T := T#30s, MON_T_STOP := T#30s, MPS :=, L_FLOW_MON :=, FLOW :=, FLOW_LL :=, FLOW_MT :=, INSTANCE := 'XA-82.01', RESTART :=, VISIBILITY :=, OPdwCmd :=, QdwState =>, QwState =>, QSTOPPING =>, QSTOP =>, QSTARTING =>, QRUN =>, QCMD_ON => "XA-82.00 OUT", QMON =>, QMON_ERR =>, QMON_T =>, QMON_T_STOP =>, QFLOW_MON =>, QFLOW_MT =>, QFLOW_ERR =>, QMPS =>, QMAN_AUT =>, QREMOTE =>, QSIM =>, QLOCK =>, QERR =>, QERR_EXT =>, QwAlarm =>)
   END_RUNG
   RUNG wire#powerrail
      Contact( "T-85.00".State.Agi_ON )
      I_Contact( #"XA-82.00".QSTOPPING )
   END_RUNG wire#w1
   // the same network as SCL:
   #"XA-82.00"(LOCK := #lock,   // "Motor"
               LIOP_SEL := #Init,
               L_AUT := #Init,
               L_REMOTE := #Init,
               L_RESET := #Reset,
               AUT_ON := "T-85.00".State.Agi_ON AND NOT #"XA-82.00".QSTOPPING,
               FB_ON := "XA-82.00 Feedback",
               L_MON := #Init,
               MON_T := T#30s,
               MON_T_STOP := T#30s,
               INSTANCE := 'XA-82.01',
               QCMD_ON => "XA-82.00 OUT");
END_REGION
END_FUNCTION_BLOCK
